    |   movel(p[0.416217, -0.000852, -0.000100, 0.000000, -3.141593, 0.000000],accel_mss,speed_ms,0,blend_radius_m)
    |   movel(p[0.416898, -0.000524, -0.000100, 0.000000, -3.141593, 0.000000],accel_mss,speed_ms,0,blend_radius_m)
    |   movel(p[0.417586, -0.000221, -0.000100, 0.000000, 3.141593, 0.000000],accel_mss,speed_ms,0,blend_radius_m)
    |   movel(p[0.417752, -0.000150, -0.000100, 0.000000, -3.141593, 0.000000],accel_mss,speed_ms,0,0.000)
    |   movel(p[0.418040, -0.000026, -0.000100, 0.000000, -3.141593, 0.000000],accel_mss,speed_ms,0,0.000)
    |   movel(p[0.418373, 0.000118, -0.000100, 0.000000, -3.141593, 0.000000],accel_mss,speed_ms,0,0.000)
    |   movel(p[0.418711, 0.000265, -0.000100, 0.000000, -3.141593, 0.000000],accel_mss,speed_ms,0,0.000)
    |   movel(p[0.419555, 0.000597, -0.000100, 0.000000, -3.141593, 0.000000],accel_mss,speed_ms,0,blend_radius_m)
    |   movel(p[0.420567, 0.000924, -0.000100, 0.000000, 3.141593, 0.000000],accel_mss,speed_ms,0,blend_radius_m)
    |   movel(p[0.421755, 0.001251, -0.000100, 0.000000, -3.141593, 0.000000],accel_mss,speed_ms,0,blend_radius_m)
    |   movel(p[0.423136, 0.001581, -0.000100, 0.000000, -3.141593, 0.000000],accel_mss,speed_ms,0,blend_radius_m)
    |   movel(p[0.424710, 0.001831, -0.000100, 0.000000, 3.141593, 0.000000],accel_mss,speed_ms,0,blend_radius_m)
    |   movel(p[0.426559, 0.001928, -0.000100, 0.000000, 3.141593, 0.000000],accel_mss,speed_ms,0,blend_radius_m)
    |   movel(p[0.428336, 0.001876, -0.000100, 0.000000, -3.141593, 0.000000],accel_mss,speed_ms,0,blend_radius_m)
    |   movel(p[0.429661, 0.001658, -0.000100, 0.000000, -3.141593, 0.000000],accel_mss,speed_ms,0,blend_radius_m)
    |   movel(p[0.430073, 0.001550, -0.000100, 0.000000, -3.141593, 0.000000],accel_mss,speed_ms,0,0.000)
    |   movel(p[0.430504, 0.001438, -0.000100, 0.000000, 3.141593, 0.000000],accel_mss,speed_ms,0,0.000)
    |   movel(p[0.430895, 0.001337, -0.000100, 0.000000, -3.141593, 0.000000],accel_mss,speed_ms,0,0.000)
    |   movel(p[0.431163, 0.001269, -0.000100, 0.000000, -3.141593, 0.000000],accel_mss,speed_ms,0,0.000)
    |   movel(p[0.432181, 0.000939, -0.000100, 0.000000, -3.141593, 0.000000],accel_mss,speed_ms,0,blend_radius_m)
    |   movel(p[0.433399, 0.000403, -0.000100, 0.000000, -3.141593, 0.000000],accel_mss,speed_ms,0,blend_radius_m)
    |   movel(p[0.434515, -0.000180, -0.000100, 0.000000, 3.141593, 0.000000],accel_mss,speed_ms,0,blend_radius_m)
    |   movel(p[0.435077, -0.000621, -0.000100, 0.000000, 3.141593, 0.000000],accel_mss,speed_ms,0,blend_radius_m)
    |   movel(p[0.435218, -0.000758, -0.000100, 0.000000, -3.141593, 0.000000],accel_mss,speed_ms,0,0.000)
    |   movel(p[0.435364, -0.000873, -0.000100, 0.000000, -3.141593, 0.000000],accel_mss,speed_ms,0,0.000)
    |   movel(p[0.435496, -0.000956, -0.000100, 0.000000, 3.141593, 0.000000],accel_mss,speed_ms,0,0.000)
    |   movel(p[0.435800, -0.001069, -0.000100, 0.000000, -3.141593, 0.000000],accel_mss,speed_ms,0,0.000)
    |   movel(p[0.437336, -0.002626, -0.000100, 0.000000, -3.141593, 0.000000],accel_mss,speed_ms,0,blend_radius_m)
    |   movel(p[0.438726, -0.004069, -0.000100, 0.000000, -3.141593, 0.000000],accel_mss,speed_ms,0,blend_radius_m)
    |   movel(p[0.439357, -0.004825, -0.000100, 0.000000, -3.141593, 0.000000],accel_mss,speed_ms,0,blend_radius_m)
    |   movel(p[0.439502, -0.005031, -0.000100, 0.000000, 3.141593, 0.000000],accel_mss,speed_ms,0,0.000)
    |   movel(p[0.439674, -0.005293, -0.000100, 0.000000, -3.141593, 0.000000],accel_mss,speed_ms,0,0.000)
    |   movel(p[0.439844, -0.005566, -0.000100, 0.000000, 3.141593, 0.000000],accel_mss,speed_ms,0,0.000)
    |   movel(p[0.439984, -0.005806, -0.000100, 0.000000, -3.141593, 0.000000],accel_mss,speed_ms,0,0.000)
    |   movel(p[0.440137, -0.006078, -0.000100, 0.000000, -3.141593, 0.000000],accel_mss,speed_ms,0,0.000)
    |   movel(p[0.440290, -0.006350, -0.000100, 0.000000, 3.141593, 0.000000],accel_mss,speed_ms,0,0.000)
    |   movel(p[0.439826, -0.006519, -0.000100, 0.000000, -3.141593, 0.000000],accel_mss,speed_ms,0,0.000)
    |   movel(p[0.439363, -0.006689, -0.000100, 0.000000, -3.141593, 0.000000],accel_mss,speed_ms,0,0.000)
    |   movel(p[0.437743, -0.007355, -0.000100, 0.000000, 3.141593, 0.000000],accel_mss,speed_ms,0,blend_radius_m)
    |   movel(p[0.436100, -0.008178, -0.000100, 0.000000, -3.141593, 0.000000],accel_mss,speed_ms,0,blend_radius_m)
    |   movel(p[0.434697, -0.009002, -0.000100, 0.000000, -3.141593, 0.000000],accel_mss,speed_ms,0,blend_radius_m)
    |   movel(p[0.434010, -0.009605, -0.000100, 0.000000, -3.141593, 0.000000],accel_mss,speed_ms,0,blend_radius_m)
    |   movel(p[0.433927, -0.009690, -0.000100, 0.000000, -3.141593, 0.000000],accel_mss,speed_ms,0,0.000)
    |   movel(p[0.433830, -0.009763, -0.000100, 0.000000, -3.141593, 0.000000],accel_mss,speed_ms,0,0.000)
    |   movel(p[0.433736, -0.009813, -0.000100, 0.000000, -3.141593, 0.000000],accel_mss,speed_ms,0,0.000)
    |   movel(p[0.433418, -0.009924, -0.000100, 0.000000, -3.141593, 0.000000],accel_mss,speed_ms,0,0.000)
    |   movel(p[0.432629, -0.010689, -0.000100, 0.000000, 3.141593, 0.000000],accel_mss,speed_ms,0,blend_radius_m)
    |   movel(p[0.431857, -0.011472, -0.000100, 0.000000, -3.141593, 0.000000],accel_mss,speed_ms,0,blend_radius_m)
    |   movel(p[0.431761, -0.011710, -0.000100, 0.000000, -3.141593, 0.000000],accel_mss,speed_ms,0,0.000)
    |   movel(p[0.431651, -0.011931, -0.000100, 0.000000, -3.141593, 0.000000],accel_mss,speed_ms,0,0.000)
    |   movel(p[0.431530, -0.012081, -0.000100, 0.000000, -3.141593, 0.000000],accel_mss,speed_ms,0,0.000)
    |   movel(p[0.431386, -0.012228, -0.000100, 0.000000, -3.141593, 0.000000],accel_mss,speed_ms,0,0.000)
    |   movel(p[0.431242, -0.012373, -0.000100, 0.000000, -3.141593, 0.000000],accel_mss,speed_ms,0,0.000)
    |   movel(p[0.431121, -0.012518, -0.000100, 0.000000, -3.141593, 0.000000],accel_mss,speed_ms,0,0.000)
    |   movel(p[0.431032, -0.012645, -0.000100, 0.000000, -3.141593, 0.000000],accel_mss,speed_ms,0,0.000)
    |   movel(p[0.430995, -0.012795, -0.000100, 0.000000, -3.141593, 0.000000],accel_mss,speed_ms,0,0.000)
    |   movel(p[0.430928, -0.012933, -0.000100, 0.000000, 3.141593, 0.000000],accel_mss,speed_ms,0,0.000)
    |   movel(p[0.430837, -0.013093, -0.000100, 0.000000, -3.141593, 0.000000],accel_mss,speed_ms,0,0.000)
    |   movel(p[0.430728, -0.013255, -0.000100, 0.000000, -3.141593, 0.000000],accel_mss,speed_ms,0,0.000)
    |   movel(p[0.430595, -0.013484, -0.000100, 0.000000, -3.141593, 0.000000],accel_mss,speed_ms,0,0.000)
    |   movel(p[0.430417, -0.013889, -0.000100, 0.000000, -3.141593, 0.000000],accel_mss,speed_ms,0,0.000)
    |   movel(p[0.430232, -0.014365, -0.000100, 0.000000, -3.141593, 0.000000],accel_mss,speed_ms,0,blend_radius_m)
    |   movel(p[0.430065, -0.014853, -0.000100, 0.000000, -3.141593, 0.000000],accel_mss,speed_ms,0,blend_radius_m)
    |   movel(p[0.429860, -0.015581, -0.000100, 0.000000, 3.141593, 0.000000],accel_mss,speed_ms,0,blend_radius_m)
    |   movel(p[0.429754, -0.016174, -0.000100, 0.000000, 3.141593, 0.000000],accel_mss,speed_ms,0,blend_radius_m)
    |   movel(p[0.429710, -0.016862, -0.000100, 0.000000, 3.141593, 0.000000],accel_mss,speed_ms,0,blend_radius_m)
    |   movel(p[0.429711, -0.017960, -0.000100, 0.000000, -3.141593, 0.000000],accel_mss,speed_ms,0,blend_radius_m)
    |   movel(p[0.429734, -0.018811, -0.000100, 0.000000, 3.141593, 0.000000],accel_mss,speed_ms,0,blend_radius_m)
    |   movel(p[0.429778, -0.019434, -0.000100, 0.000000, -3.141593, 0.000000],accel_mss,speed_ms,0,blend_radius_m)
    |   movel(p[0.429837, -0.019884, -0.000100, 0.000000, -3.141593, 0.000000],accel_mss,speed_ms,0,0.000)
    |   movel(p[0.429922, -0.020049, -0.000100, 0.000000, 3.141593, 0.000000],accel_mss,speed_ms,0,0.000)
    |   movel(p[0.430062, -0.020114, -0.000100, 0.000000, -3.141593, 0.000000],accel_mss,speed_ms,0,0.000)
    |   movel(p[0.430262, -0.020097, -0.000100, 0.000000, 3.141593, 0.000000],accel_mss,speed_ms,0,0.000)
    |   movel(p[0.430563, -0.019991, -0.000100, 0.000000, -3.141593, 0.000000],accel_mss,speed_ms,0,0.000)
    |   movel(p[0.431055, -0.019755, -0.000100, 0.000000, -3.141593, 0.000000],accel_mss,speed_ms,0,blend_radius_m)
    |   movel(p[0.431427, -0.019573, -0.000100, 0.000000, -3.141593, 0.000000],accel_mss,speed_ms,0,0.000)
    |   movel(p[0.431760, -0.019418, -0.000100, 0.000000, -3.141593, 0.000000],accel_mss,speed_ms,0,0.000)
    |   movel(p[0.432042, -0.019295, -0.000100, 0.000000, -3.141593, 0.000000],accel_mss,speed_ms,0,0.000)
    |   movel(p[0.432189, -0.019263, -0.000100, 0.000000, -3.141593, 0.000000],accel_mss,speed_ms,0,0.000)
    |   movel(p[0.432322, -0.019196, -0.000100, 0.000000, 3.141593, 0.000000],accel_mss,speed_ms,0,0.000)
    |   movel(p[0.432477, -0.019106, -0.000100, 0.000000, 3.141593, 0.000000],accel_mss,speed_ms,0,0.000)
    |   movel(p[0.432638, -0.018999, -0.000100, 0.000000, -3.141593, 0.000000],accel_mss,speed_ms,0,0.000)
    |   movel(p[0.432833, -0.018877, -0.000100, 0.000000, 3.141593, 0.000000],accel_mss,speed_ms,0,0.000)
    |   movel(p[0.433095, -0.018742, -0.000100, 0.000000, -3.141593, 0.000000],accel_mss,speed_ms,0,0.000)
    |   movel(p[0.433377, -0.018615, -0.000100, 0.000000, 3.141593, 0.000000],accel_mss,speed_ms,0,0.000)
    |   movel(p[0.433636, -0.018517, -0.000100, 0.000000, 3.141593, 0.000000],accel_mss,speed_ms,0,0.000)
    |   movel(p[0.433877, -0.018432, -0.000100, 0.000000, -3.141593, 0.000000],accel_mss,speed_ms,0,0.000)
    |   movel(p[0.434105, -0.018343, -0.000100, 0.000000, 3.141593, 0.000000],accel_mss,speed_ms,0,0.000)
    |   movel(p[0.434295, -0.018261, -0.000100, 0.000000, -3.141593, 0.000000],accel_mss,speed_ms,0,0.000)
    |   movel(p[0.434389, -0.018208, -0.000100, 0.000000, -3.141593, 0.000000],accel_mss,speed_ms,0,0.000)
    |   movel(p[0.434943, -0.017924, -0.000100, 0.000000, -3.141593, 0.000000],accel_mss,speed_ms,0,blend_radius_m)
    |   movel(p[0.436858, -0.017281, -0.000100, 0.000000, -3.141593, 0.000000],accel_mss,speed_ms,0,blend_radius_m)
    |   movel(p[0.438844, -0.016659, -0.000100, 0.000000, 3.141593, 0.000000],accel_mss,speed_ms,0,blend_radius_m)
    |   movel(p[0.440461, -0.016220, -0.000100, 0.000000, -3.141593, 0.000000],accel_mss,speed_ms,0,blend_radius_m)
    |   movel(p[0.443462, -0.015545, -0.000100, 0.000000, -3.141593, 0.000000],accel_mss,speed_ms,0,blend_radius_m)
    |   movel(p[0.445689, -0.015200, -0.000100, 0.000000, -3.141593, 0.000000],accel_mss,speed_ms,0,blend_radius_m)
    |   movel(p[0.448089, -0.015048, -0.000100, 0.000000, 3.141593, 0.000000],accel_mss,speed_ms,0,blend_radius_m)
    |   movel(p[0.451786, -0.015019, -0.000100, 0.000000, -3.141593, 0.000000],accel_mss,speed_ms,0,blend_radius_m)
    |   movel(p[0.454871, -0.015067, -0.000100, 0.000000, -3.141593, 0.000000],accel_mss,speed_ms,0,blend_radius_m)
    |   movel(p[0.456835, -0.015196, -0.000100, 0.000000, 3.141593, 0.000000],accel_mss,speed_ms,0,blend_radius_m)
    |   movel(p[0.458642, -0.015468, -0.000100, 0.000000, -3.141593, 0.000000],accel_mss,speed_ms,0,blend_radius_m)
    |   movel(p[0.461086, -0.015994, -0.000100, 0.000000, -3.141593, 0.000000],accel_mss,speed_ms,0,blend_radius_m)
    |   movel(p[0.462544, -0.016380, -0.000100, 0.000000, -3.141593, 0.000000],accel_mss,speed_ms,0,blend_radius_m)
    |   movel(p[0.464600, -0.017008, -0.000100, 0.000000, -3.141593, 0.000000],accel_mss,speed_ms,0,blend_radius_m)
    |   movel(p[0.466617, -0.017663, -0.000100, 0.000000, -3.141593, 0.000000],accel_mss,speed_ms,0,blend_radius_m)
    |   movel(p[0.467386, -0.017990, -0.000100, 0.000000, 3.141593, 0.000000],accel_mss,speed_ms,0,blend_radius_m)
    |   movel(p[0.467568, -0.018081, -0.000100, 0.000000, -3.141593, 0.000000],accel_mss,speed_ms,0,0.000)
    |   movel(p[0.467741, -0.018157, -0.000100, 0.000000, -3.141593, 0.000000],accel_mss,speed_ms,0,0.000)
    |   movel(p[0.467889, -0.018214, -0.000100, 0.000000, 3.141593, 0.000000],accel_mss,speed_ms,0,0.000)
    |   movel(p[0.468168, -0.018270, -0.000100, 0.000000, -3.141593, 0.000000],accel_mss,speed_ms,0,0.000)
    |   movel(p[0.468732, -0.018516, -0.000100, 0.000000, -3.141593, 0.000000],accel_mss,speed_ms,0,blend_radius_m)
    |   movel(p[0.469521, -0.018887, -0.000100, 0.000000, -3.141593, 0.000000],accel_mss,speed_ms,0,blend_radius_m)
    |   movel(p[0.470686, -0.019461, -0.000100, 0.000000, -3.141593, 0.000000],accel_mss,speed_ms,0,blend_radius_m)
    |   movel(p[0.472327, -0.020285, -0.000100, 0.000000, -3.141593, 0.000000],accel_mss,speed_ms,0,blend_radius_m)
    |   movel(p[0.473356, -0.020827, -0.000100, 0.000000, -3.141593, 0.000000],accel_mss,speed_ms,0,blend_radius_m)
    |   movel(p[0.474059, -0.021232, -0.000100, 0.000000, -3.141593, 0.000000],accel_mss,speed_ms,0,blend_radius_m)
    |   movel(p[0.474563, -0.021575, -0.000100, 0.000000, 3.141593, 0.000000],accel_mss,speed_ms,0,blend_radius_m)
    |   movel(p[0.474775, -0.021730, -0.000100, 0.000000, -3.141593, 0.000000],accel_mss,speed_ms,0,0.000)
    |   movel(p[0.474976, -0.021860, -0.000100, 0.000000, 3.141593, 0.000000],accel_mss,speed_ms,0,0.000)
    |   movel(p[0.475148, -0.021958, -0.000100, 0.000000, -3.141593, 0.000000],accel_mss,speed_ms,0,0.000)
    |   movel(p[0.475298, -0.021997, -0.000100, 0.000000, -3.141593, 0.000000],accel_mss,speed_ms,0,0.000)
    |   movel(p[0.475404, -0.022066, -0.000100, 0.000000, -3.141593, 0.000000],accel_mss,speed_ms,0,0.000)
    |   movel(p[0.475522, -0.022164, -0.000100, 0.000000, -3.141593, 0.000000],accel_mss,speed_ms,0,0.000)
    |   movel(p[0.475636, -0.022278, -0.000100, 0.000000, -3.141593, 0.000000],accel_mss,speed_ms,0,0.000)
    |   movel(p[0.475753, -0.022393, -0.000100, 0.000000, 3.141593, 0.000000],accel_mss,speed_ms,0,0.000)
    |   movel(p[0.475880, -0.022490, -0.000100, 0.000000, -3.141593, 0.000000],accel_mss,speed_ms,0,0.000)
    |   movel(p[0.475999, -0.022558, -0.000100, 0.000000, -3.141593, 0.000000],accel_mss,speed_ms,0,0.000)
    |   movel(p[0.476173, -0.022598, -0.000100, 0.000000, -3.141593, 0.000000],accel_mss,speed_ms,0,0.000)
    |   movel(p[0.476292, -0.022666, -0.000100, 0.000000, -3.141593, 0.000000],accel_mss,speed_ms,0,0.000)
    |   movel(p[0.476419, -0.022764, -0.000100, 0.000000, 3.141593, 0.000000],accel_mss,speed_ms,0,0.000)
    |   movel(p[0.476536, -0.022878, -0.000100, 0.000000, 3.141593, 0.000000],accel_mss,speed_ms,0,0.000)
    |   movel(p[0.476651, -0.022993, -0.000100, 0.000000, -3.141593, 0.000000],accel_mss,speed_ms,0,0.000)
    |   movel(p[0.476771, -0.023090, -0.000100, 0.000000, 3.141593, 0.000000],accel_mss,speed_ms,0,0.000)
    |   movel(p[0.476880, -0.023159, -0.000100, 0.000000, -3.141593, 0.000000],accel_mss,speed_ms,0,0.000)
    |   movel(p[0.477050, -0.023211, -0.000100, 0.000000, -3.141593, 0.000000],accel_mss,speed_ms,0,0.000)
    |   movel(p[0.477427, -0.023513, -0.000100, 0.000000, -3.141593, 0.000000],accel_mss,speed_ms,0,0.000)
    |   movel(p[0.477865, -0.023881, -0.000100, 0.000000, -3.141593, 0.000000],accel_mss,speed_ms,0,blend_radius_m)
    |   movel(p[0.478356, -0.024317, -0.000100, 0.000000, -3.141593, 0.000000],accel_mss,speed_ms,0,blend_radius_m)
    |   movel(p[0.478838, -0.024746, -0.000100, 0.000000, -3.141593, 0.000000],accel_mss,speed_ms,0,blend_radius_m)
    |   movel(p[0.479242, -0.025085, -0.000100, 0.000000, 3.141593, 0.000000],accel_mss,speed_ms,0,blend_radius_m)
    |   movel(p[0.479575, -0.025349, -0.000100, 0.000000, 3.141593, 0.000000],accel_mss,speed_ms,0,0.000)
    |   movel(p[0.480294, -0.025926, -0.000100, 0.000000, -3.141593, 0.000000],accel_mss,speed_ms,0,blend_radius_m)
    |   movel(p[0.481044, -0.026647, -0.000100, 0.000000, -3.141593, 0.000000],accel_mss,speed_ms,0,blend_radius_m)
    |   movel(p[0.481936, -0.027528, -0.000100, 0.000000, -3.141593, 0.000000],accel_mss,speed_ms,0,blend_radius_m)
    |   movel(p[0.482827, -0.028427, -0.000100, 0.000000, -3.141593, 0.000000],accel_mss,speed_ms,0,blend_radius_m)
    |   movel(p[0.483578, -0.029205, -0.000100, 0.000000, -3.141593, 0.000000],accel_mss,speed_ms,0,blend_radius_m)
    |   movel(p[0.484227, -0.029891, -0.000100, 0.000000, 3.141593, 0.000000],accel_mss,speed_ms,0,blend_radius_m)
    |   movel(p[0.484290, -0.030061, -0.000100, 0.000000, -3.141593, 0.000000],accel_mss,speed_ms,0,0.000)
    |   movel(p[0.484569, -0.030409, -0.000100, 0.000000, 3.141593, 0.000000],accel_mss,speed_ms,0,0.000)
    |   movel(p[0.484909, -0.030813, -0.000100, 0.000000, -3.141593, 0.000000],accel_mss,speed_ms,0,blend_radius_m)
    |   movel(p[0.485311, -0.031268, -0.000100, 0.000000, -3.141593, 0.000000],accel_mss,speed_ms,0,blend_radius_m)
    |   movel(p[0.485713, -0.031725, -0.000100, 0.000000, -3.141593, 0.000000],accel_mss,speed_ms,0,blend_radius_m)
    |   movel(p[0.486053, -0.032134, -0.000100, 0.000000, -3.141593, 0.000000],accel_mss,speed_ms,0,blend_radius_m)
    |   movel(p[0.486328, -0.032485, -0.000100, 0.000000, -3.141593, 0.000000],accel_mss,speed_ms,0,0.000)
    |   movel(p[0.486361, -0.032581, -0.000100, 0.000000, 3.141593, 0.000000],accel_mss,speed_ms,0,0.000)
    |   movel(p[0.486449, -0.032767, -0.000100, 0.000000, -3.141593, 0.000000],accel_mss,speed_ms,0,0.000)
    |   movel(p[0.486546, -0.032888, -0.000100, 0.000000, -3.141593, 0.000000],accel_mss,speed_ms,0,0.000)
    |   movel(p[0.486661, -0.033003, -0.000100, 0.000000, -3.141593, 0.000000],accel_mss,speed_ms,0,0.000)
    |   movel(p[0.486776, -0.033120, -0.000100, 0.000000, 3.141593, 0.000000],accel_mss,speed_ms,0,0.000)
    |   movel(p[0.486873, -0.033248, -0.000100, 0.000000, -3.141593, 0.000000],accel_mss,speed_ms,0,0.000)
    |   movel(p[0.486941, -0.033366, -0.000100, 0.000000, -3.141593, 0.000000],accel_mss,speed_ms,0,0.000)
    |   movel(p[0.486981, -0.033540, -0.000100, 0.000000, -3.141593, 0.000000],accel_mss,speed_ms,0,0.000)
    |   movel(p[0.487049, -0.033659, -0.000100, 0.000000, -3.141593, 0.000000],accel_mss,speed_ms,0,0.000)
    |   movel(p[0.487146, -0.033786, -0.000100, 0.000000, -3.141593, 0.000000],accel_mss,speed_ms,0,0.000)
    |   movel(p[0.487261, -0.033903, -0.000100, 0.000000, -3.141593, 0.000000],accel_mss,speed_ms,0,0.000)
    |   movel(p[0.487376, -0.034018, -0.000100, 0.000000, -3.141593, 0.000000],accel_mss,speed_ms,0,0.000)
    |   movel(p[0.487473, -0.034137, -0.000100, 0.000000, -3.141593, 0.000000],accel_mss,speed_ms,0,0.000)
    |   movel(p[0.487542, -0.034245, -0.000100, 0.000000, -3.141593, 0.000000],accel_mss,speed_ms,0,0.000)
    |   movel(p[0.487582, -0.034401, -0.000100, 0.000000, -3.141593, 0.000000],accel_mss,speed_ms,0,0.000)
    |   movel(p[0.487682, -0.034579, -0.000100, 0.000000, -3.141593, 0.000000],accel_mss,speed_ms,0,0.000)
    |   movel(p[0.487815, -0.034787, -0.000100, 0.000000, -3.141593, 0.000000],accel_mss,speed_ms,0,0.000)
    |   movel(p[0.487973, -0.035007, -0.000100, 0.000000, -3.141593, 0.000000],accel_mss,speed_ms,0,0.000)
    |   movel(p[0.488406, -0.035609, -0.000100, 0.000000, -3.141593, 0.000000],accel_mss,speed_ms,0,blend_radius_m)
    |   movel(p[0.488726, -0.036121, -0.000100, 0.000000, -3.141593, 0.000000],accel_mss,speed_ms,0,blend_radius_m)
    |   movel(p[0.488944, -0.036553, -0.000100, 0.000000, -3.141593, 0.000000],accel_mss,speed_ms,0,0.000)
    |   movel(p[0.489054, -0.036903, -0.000100, 0.000000, -3.141593, 0.000000],accel_mss,speed_ms,0,0.000)
    |   movel(p[0.489130, -0.037075, -0.000100, 0.000000, -3.141593, 0.000000],accel_mss,speed_ms,0,0.000)
    |   movel(p[0.489199, -0.037181, -0.000100, 0.000000, -3.141593, 0.000000],accel_mss,speed_ms,0,0.000)
    |   movel(p[0.489274, -0.037278, -0.000100, 0.000000, -3.141593, 0.000000],accel_mss,speed_ms,0,0.000)
    |   movel(p[0.489617, -0.037792, -0.000100, 0.000000, -3.141593, 0.000000],accel_mss,speed_ms,0,blend_radius_m)
    |   movel(p[0.490361, -0.039291, -0.000100, 0.000000, -3.141593, 0.000000],accel_mss,speed_ms,0,blend_radius_m)
    |   movel(p[0.491079, -0.040819, -0.000100, 0.000000, -3.141593, 0.000000],accel_mss,speed_ms,0,blend_radius_m)
    |   movel(p[0.491523, -0.041907, -0.000100, 0.000000, -3.141593, 0.000000],accel_mss,speed_ms,0,blend_radius_m)
    |   movel(p[0.492063, -0.043418, -0.000100, 0.000000, -3.141593, 0.000000],accel_mss,speed_ms,0,blend_radius_m)
    |   movel(p[0.492524, -0.044767, -0.000100, 0.000000, -3.141593, 0.000000],accel_mss,speed_ms,0,blend_radius_m)
    |   movel(p[0.492955, -0.046099, -0.000100, 0.000000, -3.141593, 0.000000],accel_mss,speed_ms,0,blend_radius_m)
    |   movel(p[0.493401, -0.047553, -0.000100, 0.000000, -3.141593, 0.000000],accel_mss,speed_ms,0,blend_radius_m)
    |   movel(p[0.493523, -0.048000, -0.000100, 0.000000, -3.141593, 0.000000],accel_mss,speed_ms,0,0.000)
    |   movel(p[0.493636, -0.048500, -0.000100, 0.000000, -3.141593, 0.000000],accel_mss,speed_ms,0,blend_radius_m)
    |   movel(p[0.493728, -0.048991, -0.000100, 0.000000, -3.141593, 0.000000],accel_mss,speed_ms,0,0.000)
    |   movel(p[0.493784, -0.049411, -0.000100, 0.000000, -3.141593, 0.000000],accel_mss,speed_ms,0,0.000)
    |   movel(p[0.493817, -0.049655, -0.000100, 0.000000, -3.141593, 0.000000],accel_mss,speed_ms,0,0.000)
    |   movel(p[0.493908, -0.050217, -0.000100, 0.000000, 3.141593, 0.000000],accel_mss,speed_ms,0,blend_radius_m)
    |   movel(p[0.494021, -0.050885, -0.000100, 0.000000, -3.141593, 0.000000],accel_mss,speed_ms,0,blend_radius_m)
    |   movel(p[0.494147, -0.051603, -0.000100, 0.000000, -3.141593, 0.000000],accel_mss,speed_ms,0,blend_radius_m)
    |   movel(p[0.494558, -0.054697, -0.000100, 0.000000, 3.141593, 0.000000],accel_mss,speed_ms,0,blend_radius_m)
    |   movel(p[0.494697, -0.057850, -0.000100, 0.000000, 3.141593, 0.000000],accel_mss,speed_ms,0,blend_radius_m)
    |   movel(p[0.494562, -0.061080, -0.000100, 0.000000, -3.141593, 0.000000],accel_mss,speed_ms,0,blend_radius_m)
    |   movel(p[0.494155, -0.064404, -0.000100, 0.000000, -3.141593, 0.000000],accel_mss,speed_ms,0,blend_radius_m)
    |   movel(p[0.494041, -0.065118, -0.000100, 0.000000, -3.141593, 0.000000],accel_mss,speed_ms,0,blend_radius_m)
    |   movel(p[0.493930, -0.065816, -0.000100, 0.000000, -3.141593, 0.000000],accel_mss,speed_ms,0,blend_radius_m)
    |   movel(p[0.493836, -0.066416, -0.000100, 0.000000, -3.141593, 0.000000],accel_mss,speed_ms,0,blend_radius_m)
    |   movel(p[0.493784, -0.066753, -0.000100, 0.000000, -3.141593, 0.000000],accel_mss,speed_ms,0,0.000)
    |   movel(p[0.493465, -0.068250, -0.000100, 0.000000, -3.141593, 0.000000],accel_mss,speed_ms,0,blend_radius_m)
    |   movel(p[0.492719, -0.070782, -0.000100, 0.000000, -3.141593, 0.000000],accel_mss,speed_ms,0,blend_radius_m)
    |   movel(p[0.491886, -0.073338, -0.000100, 0.000000, -3.141593, 0.000000],accel_mss,speed_ms,0,blend_radius_m)
    |   movel(p[0.491207, -0.075078, -0.000100, 0.000000, -3.141593, 0.000000],accel_mss,speed_ms,0,blend_radius_m)
    |   movel(p[0.491058, -0.075416, -0.000100, 0.000000, -3.141593, 0.000000],accel_mss,speed_ms,0,0.000)
    |   movel(p[0.490913, -0.075749, -0.000100, 0.000000, -3.141593, 0.000000],accel_mss,speed_ms,0,0.000)
    |   movel(p[0.490787, -0.076037, -0.000100, 0.000000, -3.141593, 0.000000],accel_mss,speed_ms,0,0.000)
    |   movel(p[0.490715, -0.076203, -0.000100, 0.000000, -3.141593, 0.000000],accel_mss,speed_ms,0,0.000)
    |   movel(p[0.490443, -0.076801, -0.000100, 0.000000, -3.141593, 0.000000],accel_mss,speed_ms,0,blend_radius_m)
    |   movel(p[0.490066, -0.077573, -0.000100, 0.000000, -3.141593, 0.000000],accel_mss,speed_ms,0,blend_radius_m)
    |   movel(p[0.489660, -0.078369, -0.000100, 0.000000, -3.141593, 0.000000],accel_mss,speed_ms,0,blend_radius_m)
    |   movel(p[0.489292, -0.079053, -0.000100, 0.000000, 3.141593, 0.000000],accel_mss,speed_ms,0,blend_radius_m)
    |   movel(p[0.489070, -0.079458, -0.000100, 0.000000, -3.141593, 0.000000],accel_mss,speed_ms,0,0.000)
    |   movel(p[0.488816, -0.079931, -0.000100, 0.000000, -3.141593, 0.000000],accel_mss,speed_ms,0,blend_radius_m)
    |   movel(p[0.488569, -0.080398, -0.000100, 0.000000, -3.141593, 0.000000],accel_mss,speed_ms,0,blend_radius_m)
    |   movel(p[0.488372, -0.080778, -0.000100, 0.000000, -3.141593, 0.000000],accel_mss,speed_ms,0,0.000)
    |   movel(p[0.488175, -0.081139, -0.000100, 0.000000, -3.141593, 0.000000],accel_mss,speed_ms,0,0.000)
    |   movel(p[0.487930, -0.081542, -0.000100, 0.000000, -3.141593, 0.000000],accel_mss,speed_ms,0,0.000)
    |   movel(p[0.487677, -0.081924, -0.000100, 0.000000, -3.141593, 0.000000],accel_mss,speed_ms,0,0.000)
    |   movel(p[0.487457, -0.082219, -0.000100, 0.000000, -3.141593, 0.000000],accel_mss,speed_ms,0,0.000)
    |   movel(p[0.487267, -0.082465, -0.000100, 0.000000, -3.141593, 0.000000],accel_mss,speed_ms,0,0.000)
    |   movel(p[0.487107, -0.082696, -0.000100, 0.000000, -3.141593, 0.000000],accel_mss,speed_ms,0,0.000)
    |   movel(p[0.486985, -0.082893, -0.000100, 0.000000, -3.141593, 0.000000],accel_mss,speed_ms,0,0.000)
    |   movel(p[0.486939, -0.083057, -0.000100, 0.000000, -3.141593, 0.000000],accel_mss,speed_ms,0,0.000)
    |   movel(p[0.486851, -0.083187, -0.000100, 0.000000, -3.141593, 0.000000],accel_mss,speed_ms,0,0.000)
    |   movel(p[0.486730, -0.083333, -0.000100, 0.000000, -3.141593, 0.000000],accel_mss,speed_ms,0,0.000)
    |   movel(p[0.486586, -0.083478, -0.000100, 0.000000, -3.141593, 0.000000],accel_mss,speed_ms,0,0.000)
    |   movel(p[0.486442, -0.083626, -0.000100, 0.000000, -3.141593, 0.000000],accel_mss,speed_ms,0,0.000)
    |   movel(p[0.486321, -0.083779, -0.000100, 0.000000, -3.141593, 0.000000],accel_mss,speed_ms,0,0.000)
    |   movel(p[0.486234, -0.083916, -0.000100, 0.000000, -3.141593, 0.000000],accel_mss,speed_ms,0,0.000)
    |   movel(p[0.486191, -0.084092, -0.000100, 0.000000, -3.141593, 0.000000],accel_mss,speed_ms,0,0.000)
    |   movel(p[0.486123, -0.084210, -0.000100, 0.000000, -3.141593, 0.000000],accel_mss,speed_ms,0,0.000)
    |   movel(p[0.486026, -0.084337, -0.000100, 0.000000, -3.141593, 0.000000],accel_mss,speed_ms,0,0.000)
    |   movel(p[0.485911, -0.084453, -0.000100, 0.000000, -3.141593, 0.000000],accel_mss,speed_ms,0,0.000)
    |   movel(p[0.485796, -0.084568, -0.000100, 0.000000, -3.141593, 0.000000],accel_mss,speed_ms,0,0.000)
    |   movel(p[0.485699, -0.084689, -0.000100, 0.000000, -3.141593, 0.000000],accel_mss,speed_ms,0,0.000)
    |   movel(p[0.485630, -0.084799, -0.000100, 0.000000, -3.141593, 0.000000],accel_mss,speed_ms,0,0.000)
    |   movel(p[0.485577, -0.084972, -0.000100, 0.000000, -3.141593, 0.000000],accel_mss,speed_ms,0,0.000)
    |   movel(p[0.485258, -0.085366, -0.000100, 0.000000, -3.141593, 0.000000],accel_mss,speed_ms,0,blend_radius_m)
    |   movel(p[0.484871, -0.085823, -0.000100, 0.000000, -3.141593, 0.000000],accel_mss,speed_ms,0,blend_radius_m)
    |   movel(p[0.484411, -0.086337, -0.000100, 0.000000, -3.141593, 0.000000],accel_mss,speed_ms,0,blend_radius_m)
    |   movel(p[0.483951, -0.086850, -0.000100, 0.000000, -3.141593, 0.000000],accel_mss,speed_ms,0,blend_radius_m)
    |   movel(p[0.483563, -0.087301, -0.000100, 0.000000, -3.141593, 0.000000],accel_mss,speed_ms,0,blend_radius_m)
    |   movel(p[0.483240, -0.087692, -0.000100, 0.000000, -3.141593, 0.000000],accel_mss,speed_ms,0,blend_radius_m)
    |   movel(p[0.483129, -0.087975, -0.000100, 0.000000, -3.141593, 0.000000],accel_mss,speed_ms,0,0.000)
    |   movel(p[0.481598, -0.089513, -0.000100, 0.000000, -3.141593, 0.000000],accel_mss,speed_ms,0,blend_radius_m)
    |   movel(p[0.480062, -0.091046, -0.000100, 0.000000, -3.141593, 0.000000],accel_mss,speed_ms,0,blend_radius_m)
    |   movel(p[0.479862, -0.091128, -0.000100, 0.000000, -3.141593, 0.000000],accel_mss,speed_ms,0,0.000)
    |   movel(p[0.479385, -0.091481, -0.000100, 0.000000, -3.141593, 0.000000],accel_mss,speed_ms,0,blend_radius_m)
    |   movel(p[0.478932, -0.091868, -0.000100, 0.000000, -3.141593, 0.000000],accel_mss,speed_ms,0,blend_radius_m)
    |   movel(p[0.478420, -0.092328, -0.000100, 0.000000, -3.141593, 0.000000],accel_mss,speed_ms,0,blend_radius_m)
    |   movel(p[0.477906, -0.092788, -0.000100, 0.000000, -3.141593, 0.000000],accel_mss,speed_ms,0,blend_radius_m)
    |   movel(p[0.477449, -0.093176, -0.000100, 0.000000, -3.141593, 0.000000],accel_mss,speed_ms,0,blend_radius_m)
    |   movel(p[0.477054, -0.093494, -0.000100, 0.000000, -3.141593, 0.000000],accel_mss,speed_ms,0,blend_radius_m)
    |   movel(p[0.476957, -0.093528, -0.000100, 0.000000, -3.141593, 0.000000],accel_mss,speed_ms,0,0.000)
    |   movel(p[0.476772, -0.093616, -0.000100, 0.000000, -3.141593, 0.000000],accel_mss,speed_ms,0,0.000)
    |   movel(p[0.476651, -0.093714, -0.000100, 0.000000, -3.141593, 0.000000],accel_mss,speed_ms,0,0.000)
    |   movel(p[0.476536, -0.093828, -0.000100, 0.000000, -3.141593, 0.000000],accel_mss,speed_ms,0,0.000)
    |   movel(p[0.476419, -0.093943, -0.000100, 0.000000, -3.141593, 0.000000],accel_mss,speed_ms,0,0.000)
    |   movel(p[0.476293, -0.094040, -0.000100, 0.000000, -3.141593, 0.000000],accel_mss,speed_ms,0,0.000)
    |   movel(p[0.476175, -0.094108, -0.000100, 0.000000, -3.141593, 0.000000],accel_mss,speed_ms,0,0.000)
    |   movel(p[0.475999, -0.094152, -0.000100, 0.000000, -3.141593, 0.000000],accel_mss,speed_ms,0,0.000)
    |   movel(p[0.475861, -0.094239, -0.000100, 0.000000, -3.141593, 0.000000],accel_mss,speed_ms,0,0.000)
    |   movel(p[0.475709, -0.094360, -0.000100, 0.000000, -3.141593, 0.000000],accel_mss,speed_ms,0,0.000)
    |   movel(p[0.475561, -0.094503, -0.000100, 0.000000, -3.141593, 0.000000],accel_mss,speed_ms,0,0.000)
    |   movel(p[0.475415, -0.094647, -0.000100, 0.000000, -3.141593, 0.000000],accel_mss,speed_ms,0,0.000)
    |   movel(p[0.475269, -0.094768, -0.000100, 0.000000, -3.141593, 0.000000],accel_mss,speed_ms,0,0.000)
    |   movel(p[0.475139, -0.094856, -0.000100, 0.000000, -3.141593, 0.000000],accel_mss,speed_ms,0,0.000)
    |   speed_ms    = 0.050
    |   movel(p[0.475139, -0.094856, 0.003000, 0.000000, -3.141593, 0.000000],accel_mss,speed_ms,0,blend_radius_m)
    |   speed_ms    = 1.000
    |   movel(p[0.475139, -0.094856, 0.015000, 0.000000, -3.141593, 0.000000],accel_mss,speed_ms,0,blend_radius_m)
    |   movel(p[0.452673, -0.050477, 0.015000, 0.000000, -3.141593, 0.000000],accel_mss,speed_ms,0,blend_radius_m)
    |   movel(p[0.452673, -0.050477, 0.003000, 0.000000, -3.141593, 0.000000],accel_mss,speed_ms,0,blend_radius_m)
    |   speed_ms    = 0.050
    |   movel(p[0.452673, -0.050477, -0.000100, 0.000000, -3.141593, 0.000000],accel_mss,speed_ms,0,blend_radius_m)
    |   speed_ms    = 0.083
    |   movel(p[0.452152, -0.050708, -0.000100, 0.000000, -3.141593, 0.000000],accel_mss,speed_ms,0,blend_radius_m)
    |   movel(p[0.451754, -0.050778, -0.000100, 0.000000, 3.141593, 0.000000],accel_mss,speed_ms,0,0.000)
    |   movel(p[0.451576, -0.050755, -0.000100, 0.000000, -3.141593, 0.000000],accel_mss,speed_ms,0,0.000)
    |   movel(p[0.451370, -0.050683, -0.000100, 0.000000, -3.141593, 0.000000],accel_mss,speed_ms,0,0.000)
    |   movel(p[0.451170, -0.050577, -0.000100, 0.000000, 3.141593, 0.000000],accel_mss,speed_ms,0,0.000)
    |   movel(p[0.451008, -0.050452, -0.000100, 0.000000, -3.141593, 0.000000],accel_mss,speed_ms,0,0.000)
    |   movel(p[0.450800, -0.050187, -0.000100, 0.000000, -3.141593, 0.000000],accel_mss,speed_ms,0,0.000)
    |   movel(p[0.450670, -0.049864, -0.000100, 0.000000, 3.141593, 0.000000],accel_mss,speed_ms,0,0.000)
    |   movel(p[0.450690, -0.049683, -0.000100, 0.000000, -3.141593, 0.000000],accel_mss,speed_ms,0,0.000)
    |   movel(p[0.450806, -0.049650, -0.000100, 0.000000, -3.141593, 0.000000],accel_mss,speed_ms,0,0.000)
    |   movel(p[0.450997, -0.049670, -0.000100, 0.000000, -3.141593, 0.000000],accel_mss,speed_ms,0,0.000)
    |   movel(p[0.451508, -0.049463, -0.000100, 0.000000, -3.141593, 0.000000],accel_mss,speed_ms,0,blend_radius_m)
    |   movel(p[0.452133, -0.049158, -0.000100, 0.000000, -3.141593, 0.000000],accel_mss,speed_ms,0,blend_radius_m)
    |   movel(p[0.452836, -0.048755, -0.000100, 0.000000, -3.141593, 0.000000],accel_mss,speed_ms,0,blend_radius_m)
    |   movel(p[0.453403, -0.048472, -0.000100, 0.000000, -3.141593, 0.000000],accel_mss,speed_ms,0,blend_radius_m)
    |   movel(p[0.453863, -0.048387, -0.000100, 0.000000, -3.141593, 0.000000],accel_mss,speed_ms,0,0.000)
    |   movel(p[0.454211, -0.048496, -0.000100, 0.000000, -3.141593, 0.000000],accel_mss,speed_ms,0,0.000)
    |   movel(p[0.454450, -0.048779, -0.000100, 0.000000, -3.141593, 0.000000],accel_mss,speed_ms,0,0.000)
    |   movel(p[0.454538, -0.048991, -0.000100, 0.000000, -3.141593, 0.000000],accel_mss,speed_ms,0,0.000)
    |   movel(p[0.454557, -0.049114, -0.000100, 0.000000, -3.141593, 0.000000],accel_mss,speed_ms,0,0.000)
    |   movel(p[0.454432, -0.049246, -0.000100, 0.000000, -3.141593, 0.000000],accel_mss,speed_ms,0,0.000)
    |   movel(p[0.454326, -0.049297, -0.000100, 0.000000, -3.141593, 0.000000],accel_mss,speed_ms,0,0.000)
    |   movel(p[0.454152, -0.049415, -0.000100, 0.000000, -3.141593, 0.000000],accel_mss,speed_ms,0,0.000)
    |   movel(p[0.453955, -0.049564, -0.000100, 0.000000, -3.141593, 0.000000],accel_mss,speed_ms,0,0.000)
    |   movel(p[0.453759, -0.049728, -0.000100, 0.000000, -3.141593, 0.000000],accel_mss,speed_ms,0,0.000)
    |   movel(p[0.453231, -0.050139, -0.000100, 0.000000, -3.141593, 0.000000],accel_mss,speed_ms,0,blend_radius_m)
    |   movel(p[0.452673, -0.050477, -0.000100, 0.000000, -3.141593, 0.000000],accel_mss,speed_ms,0,blend_radius_m)
    |   speed_ms    = 0.050
    |   movel(p[0.452673, -0.050477, 0.003000, 0.000000, -3.141593, 0.000000],accel_mss,speed_ms,0,blend_radius_m)
    |   speed_ms    = 1.000
    |   movel(p[0.452673, -0.050477, 0.015000, 0.000000, -3.141593, 0.000000],accel_mss,speed_ms,0,blend_radius_m)
    |   movel(p[0.461587, -0.045373, 0.015000, 0.000000, -3.141593, 0.000000],accel_mss,speed_ms,0,blend_radius_m)
    |   movel(p[0.461587, -0.045373, 0.003000, 0.000000, -3.141593, 0.000000],accel_mss,speed_ms,0,blend_radius_m)
    |   speed_ms    = 0.050
    |   movel(p[0.461587, -0.045373, -0.000100, 0.000000, -3.141593, 0.000000],accel_mss,speed_ms,0,blend_radius_m)
    |   speed_ms    = 0.083
    |   movel(p[0.461416, -0.044959, -0.000100, 0.000000, -3.141593, 0.000000],accel_mss,speed_ms,0,0.000)
    |   movel(p[0.461322, -0.044504, -0.000100, 0.000000, -3.141593, 0.000000],accel_mss,speed_ms,0,0.000)
    |   movel(p[0.461317, -0.044135, -0.000100, 0.000000, -3.141593, 0.000000],accel_mss,speed_ms,0,0.000)
    |   movel(p[0.461433, -0.044028, -0.000100, 0.000000, -3.141593, 0.000000],accel_mss,speed_ms,0,0.000)
    |   movel(p[0.461646, -0.044119, -0.000100, 0.000000, 3.141593, 0.000000],accel_mss,speed_ms,0,0.000)
    |   movel(p[0.461986, -0.044507, -0.000100, 0.000000, -3.141593, 0.000000],accel_mss,speed_ms,0,blend_radius_m)
    |   movel(p[0.462303, -0.044962, -0.000100, 0.000000, -3.141593, 0.000000],accel_mss,speed_ms,0,blend_radius_m)
    |   movel(p[0.462493, -0.045369, -0.000100, 0.000000, -3.141593, 0.000000],accel_mss,speed_ms,0,0.000)
    |   movel(p[0.462578, -0.045926, -0.000100, 0.000000, -3.141593, 0.000000],accel_mss,speed_ms,0,blend_radius_m)
    |   movel(p[0.462371, -0.046131, -0.000100, 0.000000, -3.141593, 0.000000],accel_mss,speed_ms,0,0.000)
    |   movel(p[0.461987, -0.045956, -0.000100, 0.000000, 3.141593, 0.000000],accel_mss,speed_ms,0,0.000)
    |   movel(p[0.461587, -0.045373, -0.000100, 0.000000, -3.141593, 0.000000],accel_mss,speed_ms,0,blend_radius_m)
    |   speed_ms    = 0.050
    |   movel(p[0.461587, -0.045373, 0.003000, 0.000000, -3.141593, 0.000000],accel_mss,speed_ms,0,blend_radius_m)
    |   speed_ms    = 1.000
    |   movel(p[0.461587, -0.045373, 0.015000, 0.000000, -3.141593, 0.000000],accel_mss,speed_ms,0,blend_radius_m)
    |   movel(p[0.458150, -0.048329, 0.015000, 0.000000, -3.141593, 0.000000],accel_mss,speed_ms,0,blend_radius_m)
    |   movel(p[0.458150, -0.048329, 0.003000, 0.000000, -3.141593, 0.000000],accel_mss,speed_ms,0,blend_radius_m)
    |   speed_ms    = 0.050
    |   movel(p[0.458150, -0.048329, -0.000100, 0.000000, -3.141593, 0.000000],accel_mss,speed_ms,0,blend_radius_m)
    |   speed_ms    = 0.083
    |   movel(p[0.458072, -0.048891, -0.000100, 0.000000, -3.141593, 0.000000],accel_mss,speed_ms,0,blend_radius_m)
    |   movel(p[0.457923, -0.049563, -0.000100, 0.000000, -3.141593, 0.000000],accel_mss,speed_ms,0,blend_radius_m)
    |   movel(p[0.457708, -0.050253, -0.000100, 0.000000, -3.141593, 0.000000],accel_mss,speed_ms,0,blend_radius_m)
    |   movel(p[0.457599, -0.050573, -0.000100, 0.000000, -3.141593, 0.000000],accel_mss,speed_ms,0,0.000)
    |   movel(p[0.457491, -0.050915, -0.000100, 0.000000, 3.141593, 0.000000],accel_mss,speed_ms,0,0.000)
    |   movel(p[0.457400, -0.051229, -0.000100, 0.000000, -3.141593, 0.000000],accel_mss,speed_ms,0,0.000)
    |   movel(p[0.457345, -0.051453, -0.000100, 0.000000, -3.141593, 0.000000],accel_mss,speed_ms,0,0.000)
    |   movel(p[0.457272, -0.051702, -0.000100, 0.000000, 3.141593, 0.000000],accel_mss,speed_ms,0,0.000)
    |   movel(p[0.457095, -0.052138, -0.000100, 0.000000, 3.141593, 0.000000],accel_mss,speed_ms,0,0.000)
    |   movel(p[0.456873, -0.052641, -0.000100, 0.000000, 3.141593, 0.000000],accel_mss,speed_ms,0,blend_radius_m)
    |   movel(p[0.456628, -0.053152, -0.000100, 0.000000, 3.141593, 0.000000],accel_mss,speed_ms,0,blend_radius_m)
    |   movel(p[0.456240, -0.053863, -0.000100, 0.000000, -3.141593, 0.000000],accel_mss,speed_ms,0,blend_radius_m)
    |   movel(p[0.455859, -0.054418, -0.000100, 0.000000, -3.141593, 0.000000],accel_mss,speed_ms,0,blend_radius_m)
    |   movel(p[0.455364, -0.054980, -0.000100, 0.000000, -3.141593, 0.000000],accel_mss,speed_ms,0,blend_radius_m)
    |   movel(p[0.454592, -0.055740, -0.000100, 0.000000, 3.141593, 0.000000],accel_mss,speed_ms,0,blend_radius_m)
    |   movel(p[0.454039, -0.056253, -0.000100, 0.000000, -3.141593, 0.000000],accel_mss,speed_ms,0,blend_radius_m)
    |   movel(p[0.453551, -0.056685, -0.000100, 0.000000, -3.141593, 0.000000],accel_mss,speed_ms,0,blend_radius_m)
    |   movel(p[0.453128, -0.057045, -0.000100, 0.000000, 3.141593, 0.000000],accel_mss,speed_ms,0,blend_radius_m)
    |   movel(p[0.452947, -0.057093, -0.000100, 0.000000, 3.141593, 0.000000],accel_mss,speed_ms,0,0.000)
    |   movel(p[0.452729, -0.057171, -0.000100, 0.000000, -3.141593, 0.000000],accel_mss,speed_ms,0,0.000)
    |   movel(p[0.452470, -0.057273, -0.000100, 0.000000, -3.141593, 0.000000],accel_mss,speed_ms,0,0.000)
    |   movel(p[0.452190, -0.057394, -0.000100, 0.000000, -3.141593, 0.000000],accel_mss,speed_ms,0,0.000)
    |   movel(p[0.451132, -0.057858, -0.000100, 0.000000, -3.141593, 0.000000],accel_mss,speed_ms,0,blend_radius_m)
    |   movel(p[0.450496, -0.058104, -0.000100, 0.000000, -3.141593, 0.000000],accel_mss,speed_ms,0,blend_radius_m)
    |   movel(p[0.449976, -0.058252, -0.000100, 0.000000, 3.141593, 0.000000],accel_mss,speed_ms,0,blend_radius_m)
    |   movel(p[0.449386, -0.058362, -0.000100, 0.000000, -3.141593, 0.000000],accel_mss,speed_ms,0,blend_radius_m)
    |   movel(p[0.449206, -0.058390, -0.000100, 0.000000, -3.141593, 0.000000],accel_mss,speed_ms,0,0.000)
    |   movel(p[0.448833, -0.058449, -0.000100, 0.000000, -3.141593, 0.000000],accel_mss,speed_ms,0,0.000)
    |   movel(p[0.448391, -0.058521, -0.000100, 0.000000, 3.141593, 0.000000],accel_mss,speed_ms,0,0.000)
    |   movel(p[0.447924, -0.058597, -0.000100, 0.000000, -3.141593, 0.000000],accel_mss,speed_ms,0,0.000)
    |   movel(p[0.447245, -0.058688, -0.000100, 0.000000, -3.141593, 0.000000],accel_mss,speed_ms,0,blend_radius_m)
    |   movel(p[0.446703, -0.058711, -0.000100, 0.000000, 3.141593, 0.000000],accel_mss,speed_ms,0,blend_radius_m)
    |   movel(p[0.446118, -0.058669, -0.000100, 0.000000, -3.141593, 0.000000],accel_mss,speed_ms,0,blend_radius_m)
    |   movel(p[0.445273, -0.058549, -0.000100, 0.000000, -3.141593, 0.000000],accel_mss,speed_ms,0,blend_radius_m)
    |   movel(p[0.444641, -0.058432, -0.000100, 0.000000, -3.141593, 0.000000],accel_mss,speed_ms,0,blend_radius_m)
    |   movel(p[0.444090, -0.058299, -0.000100, 0.000000, -3.141593, 0.000000],accel_mss,speed_ms,0,blend_radius_m)
    |   movel(p[0.443653, -0.058161, -0.000100, 0.000000, 3.141593, 0.000000],accel_mss,speed_ms,0,0.000)
    |   movel(p[0.443412, -0.058031, -0.000100, 0.000000, -3.141593, 0.000000],accel_mss,speed_ms,0,0.000)
    |   movel(p[0.443272, -0.057922, -0.000100, 0.000000, -3.141593, 0.000000],accel_mss,speed_ms,0,0.000)
    |   movel(p[0.443160, -0.057824, -0.000100, 0.000000, -3.141593, 0.000000],accel_mss,speed_ms,0,0.000)
    |   movel(p[0.443077, -0.057741, -0.000100, 0.000000, -3.141593, 0.000000],accel_mss,speed_ms,0,0.000)
    |   movel(p[0.443318, -0.057729, -0.000100, 0.000000, -3.141593, 0.000000],accel_mss,speed_ms,0,0.000)
    |   movel(p[0.443564, -0.057764, -0.000100, 0.000000, -3.141593, 0.000000],accel_mss,speed_ms,0,0.000)
    |   movel(p[0.443849, -0.057814, -0.000100, 0.000000, 3.141593, 0.000000],accel_mss,speed_ms,0,0.000)
    |   movel(p[0.445456, -0.057913, -0.000100, 0.000000, -3.141593, 0.000000],accel_mss,speed_ms,0,blend_radius_m)
    |   movel(p[0.447464, -0.057659, -0.000100, 0.000000, -3.141593, 0.000000],accel_mss,speed_ms,0,blend_radius_m)
    |   movel(p[0.449460, -0.057147, -0.000100, 0.000000, -3.141593, 0.000000],accel_mss,speed_ms,0,blend_radius_m)
    |   movel(p[0.451036, -0.056444, -0.000100, 0.000000, -3.141593, 0.000000],accel_mss,speed_ms,0,blend_radius_m)
    |   movel(p[0.451197, -0.056354, -0.000100, 0.000000, -3.141593, 0.000000],accel_mss,speed_ms,0,0.000)
    |   movel(p[0.451454, -0.056217, -0.000100, 0.000000, -3.141593, 0.000000],accel_mss,speed_ms,0,0.000)
    |   movel(p[0.451746, -0.056065, -0.000100, 0.000000, -3.141593, 0.000000],accel_mss,speed_ms,0,0.000)
    |   movel(p[0.452036, -0.055917, -0.000100, 0.000000, -3.141593, 0.000000],accel_mss,speed_ms,0,0.000)
    |   movel(p[0.452317, -0.055766, -0.000100, 0.000000, -3.141593, 0.000000],accel_mss,speed_ms,0,0.000)
    |   movel(p[0.452584, -0.055604, -0.000100, 0.000000, -3.141593, 0.000000],accel_mss,speed_ms,0,0.000)
    |   movel(p[0.452804, -0.055452, -0.000100, 0.000000, -3.141593, 0.000000],accel_mss,speed_ms,0,0.000)
    |   movel(p[0.452917, -0.055346, -0.000100, 0.000000, -3.141593, 0.000000],accel_mss,speed_ms,0,0.000)
    |   movel(p[0.452999, -0.055263, -0.000100, 0.000000, -3.141593, 0.000000],accel_mss,speed_ms,0,0.000)
    |   movel(p[0.453096, -0.055192, -0.000100, 0.000000, -3.141593, 0.000000],accel_mss,speed_ms,0,0.000)
    |   movel(p[0.453192, -0.055144, -0.000100, 0.000000, 3.141593, 0.000000],accel_mss,speed_ms,0,0.000)
    |   movel(p[0.453506, -0.055035, -0.000100, 0.000000, -3.141593, 0.000000],accel_mss,speed_ms,0,0.000)
    |   movel(p[0.454231, -0.054329, -0.000100, 0.000000, -3.141593, 0.000000],accel_mss,speed_ms,0,blend_radius_m)
    |   movel(p[0.454909, -0.053619, -0.000100, 0.000000, -3.141593, 0.000000],accel_mss,speed_ms,0,blend_radius_m)
    |   movel(p[0.455244, -0.053159, -0.000100, 0.000000, -3.141593, 0.000000],accel_mss,speed_ms,0,blend_radius_m)
    |   movel(p[0.455333, -0.053000, -0.000100, 0.000000, -3.141593, 0.000000],accel_mss,speed_ms,0,0.000)
    |   movel(p[0.455430, -0.052818, -0.000100, 0.000000, -3.141593, 0.000000],accel_mss,speed_ms,0,0.000)
    |   movel(p[0.455520, -0.052640, -0.000100, 0.000000, -3.141593, 0.000000],accel_mss,speed_ms,0,0.000)
    |   movel(p[0.455589, -0.052497, -0.000100, 0.000000, -3.141593, 0.000000],accel_mss,speed_ms,0,0.000)
    |   movel(p[0.455660, -0.052365, -0.000100, 0.000000, -3.141593, 0.000000],accel_mss,speed_ms,0,0.000)
    |   movel(p[0.455759, -0.052222, -0.000100, 0.000000, -3.141593, 0.000000],accel_mss,speed_ms,0,0.000)
    |   movel(p[0.455868, -0.052090, -0.000100, 0.000000, -3.141593, 0.000000],accel_mss,speed_ms,0,0.000)
    |   movel(p[0.455970, -0.051991, -0.000100, 0.000000, -3.141593, 0.000000],accel_mss,speed_ms,0,0.000)
    |   movel(p[0.456062, -0.051895, -0.000100, 0.000000, -3.141593, 0.000000],accel_mss,speed_ms,0,0.000)
    |   movel(p[0.456140, -0.051770, -0.000100, 0.000000, 3.141593, 0.000000],accel_mss,speed_ms,0,0.000)
    |   movel(p[0.456193, -0.051638, -0.000100, 0.000000, 3.141593, 0.000000],accel_mss,speed_ms,0,0.000)
    |   movel(p[0.456211, -0.051519, -0.000100, 0.000000, 3.141593, 0.000000],accel_mss,speed_ms,0,0.000)
    |   movel(p[0.456222, -0.051408, -0.000100, 0.000000, -3.141593, 0.000000],accel_mss,speed_ms,0,0.000)
    |   movel(p[0.456254, -0.051300, -0.000100, 0.000000, -3.141593, 0.000000],accel_mss,speed_ms,0,0.000)
    |   movel(p[0.456301, -0.051210, -0.000100, 0.000000, 3.141593, 0.000000],accel_mss,speed_ms,0,0.000)
    |   movel(p[0.456437, -0.051075, -0.000100, 0.000000, -3.141593, 0.000000],accel_mss,speed_ms,0,0.000)
    |   movel(p[0.456627, -0.050757, -0.000100, 0.000000, -3.141593, 0.000000],accel_mss,speed_ms,0,0.000)
    |   movel(p[0.456842, -0.050369, -0.000100, 0.000000, -3.141593, 0.000000],accel_mss,speed_ms,0,0.000)
    |   movel(p[0.457070, -0.049927, -0.000100, 0.000000, -3.141593, 0.000000],accel_mss,speed_ms,0,0.000)
    |   movel(p[0.457612, -0.048842, -0.000100, 0.000000, -3.141593, 0.000000],accel_mss,speed_ms,0,blend_radius_m)
    |   movel(p[0.457818, -0.048462, -0.000100, 0.000000, -3.141593, 0.000000],accel_mss,speed_ms,0,0.000)
    |   movel(p[0.457947, -0.048280, -0.000100, 0.000000, -3.141593, 0.000000],accel_mss,speed_ms,0,0.000)
    |   movel(p[0.458060, -0.048228, -0.000100, 0.000000, -3.141593, 0.000000],accel_mss,speed_ms,0,0.000)
    |   movel(p[0.458150, -0.048329, -0.000100, 0.000000, -3.141593, 0.000000],accel_mss,speed_ms,0,0.000)
    |   speed_ms    = 0.050
    |   movel(p[0.458150, -0.048329, 0.003000, 0.000000, -3.141593, 0.000000],accel_mss,speed_ms,0,blend_radius_m)
    |   speed_ms    = 1.000
    |   movel(p[0.458150, -0.048329, 0.015000, 0.000000, -3.141593, 0.000000],accel_mss,speed_ms,0,blend_radius_m)
    |   movel(p[0.460013, -0.046384, 0.015000, 0.000000, -3.141593, 0.000000],accel_mss,speed_ms,0,blend_radius_m)
    |   movel(p[0.460013, -0.046384, 0.003000, 0.000000, -3.141593, 0.000000],accel_mss,speed_ms,0,blend_radius_m)
    |   speed_ms    = 0.050
    |   movel(p[0.460013, -0.046384, -0.000100, 0.000000, -3.141593, 0.000000],accel_mss,speed_ms,0,blend_radius_m)
    |   speed_ms    = 0.083
    |   movel(p[0.459961, -0.046278, -0.000100, 0.000000, -3.141593, 0.000000],accel_mss,speed_ms,0,0.000)
    |   movel(p[0.460025, -0.046172, -0.000100, 0.000000, 3.141593, 0.000000],accel_mss,speed_ms,0,0.000)
    |   movel(p[0.460180, -0.046128, -0.000100, 0.000000, -3.141593, 0.000000],accel_mss,speed_ms,0,0.000)
    |   movel(p[0.460462, -0.046184, -0.000100, 0.000000, 3.141593, 0.000000],accel_mss,speed_ms,0,0.000)
    |   movel(p[0.460926, -0.046394, -0.000100, 0.000000, -3.141593, 0.000000],accel_mss,speed_ms,0,blend_radius_m)
    |   movel(p[0.461377, -0.046637, -0.000100, 0.000000, -3.141593, 0.000000],accel_mss,speed_ms,0,blend_radius_m)
    |   movel(p[0.461457, -0.046771, -0.000100, 0.000000, -3.141593, 0.000000],accel_mss,speed_ms,0,0.000)
    |   movel(p[0.461379, -0.046920, -0.000100, 0.000000, -3.141593, 0.000000],accel_mss,speed_ms,0,0.000)
    |   movel(p[0.461177, -0.046976, -0.000100, 0.000000, -3.141593, 0.000000],accel_mss,speed_ms,0,0.000)
    |   movel(p[0.460904, -0.046913, -0.000100, 0.000000, -3.141593, 0.000000],accel_mss,speed_ms,0,0.000)
    |   movel(p[0.460656, -0.046747, -0.000100, 0.000000, 3.141593, 0.000000],accel_mss,speed_ms,0,0.000)
    |   movel(p[0.460513, -0.046625, -0.000100, 0.000000, -3.141593, 0.000000],accel_mss,speed_ms,0,0.000)
    |   movel(p[0.460364, -0.046522, -0.000100, 0.000000, -3.141593, 0.000000],accel_mss,speed_ms,0,0.000)
    |   movel(p[0.460229, -0.046449, -0.000100, 0.000000, -3.141593, 0.000000],accel_mss,speed_ms,0,0.000)
    |   movel(p[0.460071, -0.046417, -0.000100, 0.000000, -3.141593, 0.000000],accel_mss,speed_ms,0,0.000)
    |   speed_ms    = 0.050
    |   movel(p[0.460013, -0.046384, 0.003000, 0.000000, -3.141593, 0.000000],accel_mss,speed_ms,0,blend_radius_m)
    |   speed_ms    = 1.000
    |   movel(p[0.460013, -0.046384, 0.015000, 0.000000, -3.141593, 0.000000],accel_mss,speed_ms,0,blend_radius_m)
    |   movel(p[0.460275, -0.045372, 0.015000, 0.000000, -3.141593, 0.000000],accel_mss,speed_ms,0,blend_radius_m)
    |   movel(p[0.460275, -0.045372, 0.003000, 0.000000, -3.141593, 0.000000],accel_mss,speed_ms,0,blend_radius_m)
    |   speed_ms    = 0.050
    |   movel(p[0.460275, -0.045372, -0.000100, 0.000000, -3.141593, 0.000000],accel_mss,speed_ms,0,blend_radius_m)
    |   speed_ms    = 0.083
    |   movel(p[0.459823, -0.045339, -0.000100, 0.000000, 3.141593, 0.000000],accel_mss,speed_ms,0,0.000)
    |   movel(p[0.459426, -0.045318, -0.000100, 0.000000, -3.141593, 0.000000],accel_mss,speed_ms,0,0.000)
    |   movel(p[0.459076, -0.045329, -0.000100, 0.000000, 3.141593, 0.000000],accel_mss,speed_ms,0,0.000)
    |   movel(p[0.458787, -0.045370, -0.000100, 0.000000, -3.141593, 0.000000],accel_mss,speed_ms,0,0.000)
    |   movel(p[0.458582, -0.045442, -0.000100, 0.000000, -3.141593, 0.000000],accel_mss,speed_ms,0,0.000)
    |   movel(p[0.458309, -0.045545, -0.000100, 0.000000, -3.141593, 0.000000],accel_mss,speed_ms,0,0.000)
    |   movel(p[0.458061, -0.045557, -0.000100, 0.000000, -3.141593, 0.000000],accel_mss,speed_ms,0,0.000)
    |   movel(p[0.457819, -0.045476, -0.000100, 0.000000, -3.141593, 0.000000],accel_mss,speed_ms,0,0.000)
    |   movel(p[0.457561, -0.045298, -0.000100, 0.000000, -3.141593, 0.000000],accel_mss,speed_ms,0,0.000)
    |   movel(p[0.457413, -0.045191, -0.000100, 0.000000, -3.141593, 0.000000],accel_mss,speed_ms,0,0.000)
    |   movel(p[0.457055, -0.044980, -0.000100, 0.000000, 3.141593, 0.000000],accel_mss,speed_ms,0,0.000)
    |   movel(p[0.456624, -0.044738, -0.000100, 0.000000, -3.141593, 0.000000],accel_mss,speed_ms,0,0.000)
    |   movel(p[0.456156, -0.044487, -0.000100, 0.000000, -3.141593, 0.000000],accel_mss,speed_ms,0,blend_radius_m)
    |   movel(p[0.454347, -0.043738, -0.000100, 0.000000, -3.141593, 0.000000],accel_mss,speed_ms,0,blend_radius_m)
    |   movel(p[0.452107, -0.043177, -0.000100, 0.000000, 3.141593, 0.000000],accel_mss,speed_ms,0,blend_radius_m)
    |   movel(p[0.449872, -0.042876, -0.000100, 0.000000, -3.141593, 0.000000],accel_mss,speed_ms,0,blend_radius_m)
    |   movel(p[0.448094, -0.042938, -0.000100, 0.000000, -3.141593, 0.000000],accel_mss,speed_ms,0,blend_radius_m)
    |   movel(p[0.446696, -0.043209, -0.000100, 0.000000, -3.141593, 0.000000],accel_mss,speed_ms,0,blend_radius_m)
    |   movel(p[0.445440, -0.043586, -0.000100, 0.000000, 3.141593, 0.000000],accel_mss,speed_ms,0,blend_radius_m)
    |   movel(p[0.444430, -0.044025, -0.000100, 0.000000, -3.141593, 0.000000],accel_mss,speed_ms,0,blend_radius_m)
    |   movel(p[0.443832, -0.044484, -0.000100, 0.000000, -3.141593, 0.000000],accel_mss,speed_ms,0,blend_radius_m)
    |   movel(p[0.443694, -0.044619, -0.000100, 0.000000, -3.141593, 0.000000],accel_mss,speed_ms,0,0.000)
    |   movel(p[0.443523, -0.044754, -0.000100, 0.000000, -3.141593, 0.000000],accel_mss,speed_ms,0,0.000)
    |   movel(p[0.443347, -0.044870, -0.000100, 0.000000, -3.141593, 0.000000],accel_mss,speed_ms,0,0.000)
    |   movel(p[0.443196, -0.044943, -0.000100, 0.000000, -3.141593, 0.000000],accel_mss,speed_ms,0,0.000)
    |   movel(p[0.443056, -0.045018, -0.000100, 0.000000, -3.141593, 0.000000],accel_mss,speed_ms,0,0.000)
    |   movel(p[0.442917, -0.045135, -0.000100, 0.000000, -3.141593, 0.000000],accel_mss,speed_ms,0,0.000)
    |   movel(p[0.442800, -0.045273, -0.000100, 0.000000, -3.141593, 0.000000],accel_mss,speed_ms,0,0.000)
    |   movel(p[0.442725, -0.045413, -0.000100, 0.000000, -3.141593, 0.000000],accel_mss,speed_ms,0,0.000)
    |   movel(p[0.442652, -0.045565, -0.000100, 0.000000, -3.141593, 0.000000],accel_mss,speed_ms,0,0.000)
    |   movel(p[0.442537, -0.045740, -0.000100, 0.000000, -3.141593, 0.000000],accel_mss,speed_ms,0,0.000)
    |   movel(p[0.442402, -0.045911, -0.000100, 0.000000, -3.141593, 0.000000],accel_mss,speed_ms,0,0.000)
    |   movel(p[0.442267, -0.046050, -0.000100, 0.000000, -3.141593, 0.000000],accel_mss,speed_ms,0,0.000)
    |   movel(p[0.442029, -0.046325, -0.000100, 0.000000, 3.141593, 0.000000],accel_mss,speed_ms,0,0.000)
    |   movel(p[0.441763, -0.046766, -0.000100, 0.000000, -3.141593, 0.000000],accel_mss,speed_ms,0,blend_radius_m)
    |   movel(p[0.441487, -0.047332, -0.000100, 0.000000, -3.141593, 0.000000],accel_mss,speed_ms,0,blend_radius_m)
    |   movel(p[0.441211, -0.048003, -0.000100, 0.000000, -3.141593, 0.000000],accel_mss,speed_ms,0,blend_radius_m)
    |   movel(p[0.441009, -0.048282, -0.000100, 0.000000, 3.141593, 0.000000],accel_mss,speed_ms,0,0.000)
    |   movel(p[0.440736, -0.048344, -0.000100, 0.000000, 3.141593, 0.000000],accel_mss,speed_ms,0,0.000)
    |   movel(p[0.440366, -0.048161, -0.000100, 0.000000, -3.141593, 0.000000],accel_mss,speed_ms,0,0.000)
    |   movel(p[0.439855, -0.047690, -0.000100, 0.000000, -3.141593, 0.000000],accel_mss,speed_ms,0,blend_radius_m)
    |   movel(p[0.439577, -0.047416, -0.000100, 0.000000, -3.141593, 0.000000],accel_mss,speed_ms,0,0.000)
    |   movel(p[0.439294, -0.047162, -0.000100, 0.000000, -3.141593, 0.000000],accel_mss,speed_ms,0,0.000)
    |   movel(p[0.439043, -0.046958, -0.000100, 0.000000, -3.141593, 0.000000],accel_mss,speed_ms,0,0.000)
    |   movel(p[0.438886, -0.046862, -0.000100, 0.000000, -3.141593, 0.000000],accel_mss,speed_ms,0,0.000)
    |   movel(p[0.438740, -0.046789, -0.000100, 0.000000, 3.141593, 0.000000],accel_mss,speed_ms,0,0.000)
    |   movel(p[0.438542, -0.046678, -0.000100, 0.000000, -3.141593, 0.000000],accel_mss,speed_ms,0,0.000)
    |   movel(p[0.438330, -0.046551, -0.000100, 0.000000, -3.141593, 0.000000],accel_mss,speed_ms,0,0.000)
    |   movel(p[0.438136, -0.046428, -0.000100, 0.000000, -3.141593, 0.000000],accel_mss,speed_ms,0,0.000)
    |   movel(p[0.437421, -0.046004, -0.000100, 0.000000, -3.141593, 0.000000],accel_mss,speed_ms,0,blend_radius_m)
    |   movel(p[0.436390, -0.045479, -0.000100, 0.000000, -3.141593, 0.000000],accel_mss,speed_ms,0,blend_radius_m)
    |   movel(p[0.435364, -0.044995, -0.000100, 0.000000, -3.141593, 0.000000],accel_mss,speed_ms,0,blend_radius_m)
    |   movel(p[0.434919, -0.044861, -0.000100, 0.000000, 3.141593, 0.000000],accel_mss,speed_ms,0,0.000)
    |   movel(p[0.433354, -0.044623, -0.000100, 0.000000, -3.141593, 0.000000],accel_mss,speed_ms,0,blend_radius_m)
    |   movel(p[0.432422, -0.044522, -0.000100, 0.000000, 3.141593, 0.000000],accel_mss,speed_ms,0,blend_radius_m)
    |   movel(p[0.431635, -0.044500, -0.000100, 0.000000, -3.141593, 0.000000],accel_mss,speed_ms,0,blend_radius_m)
    |   movel(p[0.430668, -0.044543, -0.000100, 0.000000, -3.141593, 0.000000],accel_mss,speed_ms,0,blend_radius_m)
    |   movel(p[0.430059, -0.044587, -0.000100, 0.000000, -3.141593, 0.000000],accel_mss,speed_ms,0,blend_radius_m)
    |   movel(p[0.429498, -0.044631, -0.000100, 0.000000, -3.141593, 0.000000],accel_mss,speed_ms,0,blend_radius_m)
    |   movel(p[0.429027, -0.044670, -0.000100, 0.000000, -3.141593, 0.000000],accel_mss,speed_ms,0,0.000)
    |   movel(p[0.428836, -0.044691, -0.000100, 0.000000, -3.141593, 0.000000],accel_mss,speed_ms,0,0.000)
    |   movel(p[0.427123, -0.045042, -0.000100, 0.000000, -3.141593, 0.000000],accel_mss,speed_ms,0,blend_radius_m)
    |   movel(p[0.425657, -0.045602, -0.000100, 0.000000, -3.141593, 0.000000],accel_mss,speed_ms,0,blend_radius_m)
    |   movel(p[0.424330, -0.046426, -0.000100, 0.000000, -3.141593, 0.000000],accel_mss,speed_ms,0,blend_radius_m)
    |   movel(p[0.423032, -0.047566, -0.000100, 0.000000, -3.141593, 0.000000],accel_mss,speed_ms,0,blend_radius_m)
    |   movel(p[0.422546, -0.048049, -0.000100, 0.000000, -3.141593, 0.000000],accel_mss,speed_ms,0,blend_radius_m)
    |   movel(p[0.422119, -0.048457, -0.000100, 0.000000, 3.141593, 0.000000],accel_mss,speed_ms,0,blend_radius_m)
    |   movel(p[0.421747, -0.048799, -0.000100, 0.000000, -3.141593, 0.000000],accel_mss,speed_ms,0,blend_radius_m)
    |   movel(p[0.421587, -0.048770, -0.000100, 0.000000, -3.141593, 0.000000],accel_mss,speed_ms,0,0.000)
    |   movel(p[0.421592, -0.048648, -0.000100, 0.000000, -3.141593, 0.000000],accel_mss,speed_ms,0,0.000)
    |   movel(p[0.421735, -0.048438, -0.000100, 0.000000, -3.141593, 0.000000],accel_mss,speed_ms,0,0.000)
    |   movel(p[0.422011, -0.048153, -0.000100, 0.000000, -3.141593, 0.000000],accel_mss,speed_ms,0,0.000)
    |   movel(p[0.422183, -0.047978, -0.000100, 0.000000, -3.141593, 0.000000],accel_mss,speed_ms,0,0.000)
    |   movel(p[0.422329, -0.047806, -0.000100, 0.000000, 3.141593, 0.000000],accel_mss,speed_ms,0,0.000)
    |   movel(p[0.422437, -0.047656, -0.000100, 0.000000, -3.141593, 0.000000],accel_mss,speed_ms,0,0.000)
    |   movel(p[0.422586, -0.047251, -0.000100, 0.000000, -3.141593, 0.000000],accel_mss,speed_ms,0,0.000)
    |   movel(p[0.424352, -0.045326, -0.000100, 0.000000, -3.141593, 0.000000],accel_mss,speed_ms,0,blend_radius_m)
    |   movel(p[0.426139, -0.043405, -0.000100, 0.000000, -3.141593, 0.000000],accel_mss,speed_ms,0,blend_radius_m)
    |   movel(p[0.426430, -0.043278, -0.000100, 0.000000, -3.141593, 0.000000],accel_mss,speed_ms,0,0.000)
    |   movel(p[0.426529, -0.043245, -0.000100, 0.000000, -3.141593, 0.000000],accel_mss,speed_ms,0,0.000)
    |   movel(p[0.426765, -0.043058, -0.000100, 0.000000, -3.141593, 0.000000],accel_mss,speed_ms,0,0.000)
    |   movel(p[0.427041, -0.042816, -0.000100, 0.000000, 3.141593, 0.000000],accel_mss,speed_ms,0,0.000)
    |   movel(p[0.427336, -0.042528, -0.000100, 0.000000, 3.141593, 0.000000],accel_mss,speed_ms,0,0.000)
    |   movel(p[0.427629, -0.042241, -0.000100, 0.000000, 3.141593, 0.000000],accel_mss,speed_ms,0,0.000)
    |   movel(p[0.427897, -0.041999, -0.000100, 0.000000, -3.141593, 0.000000],accel_mss,speed_ms,0,0.000)
    |   movel(p[0.428128, -0.041807, -0.000100, 0.000000, -3.141593, 0.000000],accel_mss,speed_ms,0,0.000)
    |   movel(p[0.428295, -0.041752, -0.000100, 0.000000, 3.141593, 0.000000],accel_mss,speed_ms,0,0.000)
    |   movel(p[0.428554, -0.041566, -0.000100, 0.000000, -3.141593, 0.000000],accel_mss,speed_ms,0,0.000)
    |   movel(p[0.428857, -0.041333, -0.000100, 0.000000, -3.141593, 0.000000],accel_mss,speed_ms,0,0.000)
    |   movel(p[0.429191, -0.041056, -0.000100, 0.000000, -3.141593, 0.000000],accel_mss,speed_ms,0,0.000)
    |   movel(p[0.429555, -0.040761, -0.000100, 0.000000, -3.141593, 0.000000],accel_mss,speed_ms,0,0.000)
    |   movel(p[0.429951, -0.040471, -0.000100, 0.000000, -3.141593, 0.000000],accel_mss,speed_ms,0,0.000)
    |   movel(p[0.430321, -0.040225, -0.000100, 0.000000, -3.141593, 0.000000],accel_mss,speed_ms,0,0.000)
    |   movel(p[0.430592, -0.040077, -0.000100, 0.000000, -3.141593, 0.000000],accel_mss,speed_ms,0,0.000)
    |   movel(p[0.430811, -0.039969, -0.000100, 0.000000, -3.141593, 0.000000],accel_mss,speed_ms,0,0.000)
    |   movel(p[0.431010, -0.039856, -0.000100, 0.000000, 3.141593, 0.000000],accel_mss,speed_ms,0,0.000)
    |   movel(p[0.431169, -0.039751, -0.000100, 0.000000, 3.141593, 0.000000],accel_mss,speed_ms,0,0.000)
    |   movel(p[0.431290, -0.039618, -0.000100, 0.000000, -3.141593, 0.000000],accel_mss,speed_ms,0,0.000)
    |   movel(p[0.431412, -0.039525, -0.000100, 0.000000, 3.141593, 0.000000],accel_mss,speed_ms,0,0.000)
    |   movel(p[0.431563, -0.039425, -0.000100, 0.000000, -3.141593, 0.000000],accel_mss,speed_ms,0,0.000)
    |   movel(p[0.431726, -0.039333, -0.000100, 0.000000, -3.141593, 0.000000],accel_mss,speed_ms,0,0.000)
    |   movel(p[0.431960, -0.039211, -0.000100, 0.000000, -3.141593, 0.000000],accel_mss,speed_ms,0,0.000)
    |   movel(p[0.432390, -0.038985, -0.000100, 0.000000, -3.141593, 0.000000],accel_mss,speed_ms,0,0.000)
    |   movel(p[0.432893, -0.038720, -0.000100, 0.000000, -3.141593, 0.000000],accel_mss,speed_ms,0,blend_radius_m)
    |   movel(p[0.433412, -0.038448, -0.000100, 0.000000, 3.141593, 0.000000],accel_mss,speed_ms,0,blend_radius_m)
    |   movel(p[0.433944, -0.038176, -0.000100, 0.000000, -3.141593, 0.000000],accel_mss,speed_ms,0,blend_radius_m)
    |   movel(p[0.434489, -0.037916, -0.000100, 0.000000, -3.141593, 0.000000],accel_mss,speed_ms,0,blend_radius_m)
    |   movel(p[0.434973, -0.037700, -0.000100, 0.000000, 3.141593, 0.000000],accel_mss,speed_ms,0,blend_radius_m)
    |   movel(p[0.435287, -0.037583, -0.000100, 0.000000, -3.141593, 0.000000],accel_mss,speed_ms,0,0.000)
    |   movel(p[0.435527, -0.037500, -0.000100, 0.000000, -3.141593, 0.000000],accel_mss,speed_ms,0,0.000)
    |   movel(p[0.435754, -0.037414, -0.000100, 0.000000, -3.141593, 0.000000],accel_mss,speed_ms,0,0.000)
    |   movel(p[0.435943, -0.037333, -0.000100, 0.000000, -3.141593, 0.000000],accel_mss,speed_ms,0,0.000)
    |   movel(p[0.436036, -0.037279, -0.000100, 0.000000, 3.141593, 0.000000],accel_mss,speed_ms,0,0.000)
    |   movel(p[0.436379, -0.037098, -0.000100, 0.000000, -3.141593, 0.000000],accel_mss,speed_ms,0,0.000)
    |   movel(p[0.437384, -0.036765, -0.000100, 0.000000, 3.141593, 0.000000],accel_mss,speed_ms,0,blend_radius_m)
    |   movel(p[0.438577, -0.036405, -0.000100, 0.000000, -3.141593, 0.000000],accel_mss,speed_ms,0,blend_radius_m)
    |   movel(p[0.439861, -0.036058, -0.000100, 0.000000, 3.141593, 0.000000],accel_mss,speed_ms,0,blend_radius_m)
    |   movel(p[0.443288, -0.035424, -0.000100, 0.000000, -3.141593, 0.000000],accel_mss,speed_ms,0,blend_radius_m)
    |   movel(p[0.447124, -0.035178, -0.000100, 0.000000, -3.141593, 0.000000],accel_mss,speed_ms,0,blend_radius_m)
    |   movel(p[0.451004, -0.035322, -0.000100, 0.000000, -3.141593, 0.000000],accel_mss,speed_ms,0,blend_radius_m)
    |   movel(p[0.454561, -0.035863, -0.000100, 0.000000, -3.141593, 0.000000],accel_mss,speed_ms,0,blend_radius_m)
    |   movel(p[0.456004, -0.036199, -0.000100, 0.000000, -3.141593, 0.000000],accel_mss,speed_ms,0,blend_radius_m)
    |   movel(p[0.457480, -0.036584, -0.000100, 0.000000, -3.141593, 0.000000],accel_mss,speed_ms,0,blend_radius_m)
    |   movel(p[0.458827, -0.036962, -0.000100, 0.000000, -3.141593, 0.000000],accel_mss,speed_ms,0,blend_radius_m)
    |   movel(p[0.459132, -0.037118, -0.000100, 0.000000, -3.141593, 0.000000],accel_mss,speed_ms,0,0.000)
    |   movel(p[0.459227, -0.037176, -0.000100, 0.000000, -3.141593, 0.000000],accel_mss,speed_ms,0,0.000)
    |   movel(p[0.459417, -0.037260, -0.000100, 0.000000, -3.141593, 0.000000],accel_mss,speed_ms,0,0.000)
    |   movel(p[0.459645, -0.037348, -0.000100, 0.000000, -3.141593, 0.000000],accel_mss,speed_ms,0,0.000)
    |   movel(p[0.459886, -0.037430, -0.000100, 0.000000, -3.141593, 0.000000],accel_mss,speed_ms,0,0.000)
    |   movel(p[0.460780, -0.037778, -0.000100, 0.000000, -3.141593, 0.000000],accel_mss,speed_ms,0,blend_radius_m)
    |   movel(p[0.462551, -0.038624, -0.000100, 0.000000, 3.141593, 0.000000],accel_mss,speed_ms,0,blend_radius_m)
    |   movel(p[0.464319, -0.039507, -0.000100, 0.000000, -3.141593, 0.000000],accel_mss,speed_ms,0,blend_radius_m)
    |   movel(p[0.465000, -0.039931, -0.000100, 0.000000, 3.141593, 0.000000],accel_mss,speed_ms,0,blend_radius_m)
    |   movel(p[0.465189, -0.040064, -0.000100, 0.000000, 3.141593, 0.000000],accel_mss,speed_ms,0,0.000)
    |   movel(p[0.465372, -0.040176, -0.000100, 0.000000, -3.141593, 0.000000],accel_mss,speed_ms,0,0.000)
    |   movel(p[0.465530, -0.040259, -0.000100, 0.000000, -3.141593, 0.000000],accel_mss,speed_ms,0,0.000)
    |   movel(p[0.465690, -0.040298, -0.000100, 0.000000, -3.141593, 0.000000],accel_mss,speed_ms,0,0.000)
    |   movel(p[0.465800, -0.040366, -0.000100, 0.000000, -3.141593, 0.000000],accel_mss,speed_ms,0,0.000)
    |   movel(p[0.465921, -0.040464, -0.000100, 0.000000, -3.141593, 0.000000],accel_mss,speed_ms,0,0.000)
    |   movel(p[0.466036, -0.040578, -0.000100, 0.000000, -3.141593, 0.000000],accel_mss,speed_ms,0,0.000)
    |   movel(p[0.466153, -0.040693, -0.000100, 0.000000, -3.141593, 0.000000],accel_mss,speed_ms,0,0.000)
    |   movel(p[0.466279, -0.040790, -0.000100, 0.000000, -3.141593, 0.000000],accel_mss,speed_ms,0,0.000)
    |   movel(p[0.466397, -0.040858, -0.000100, 0.000000, -3.141593, 0.000000],accel_mss,speed_ms,0,0.000)
    |   movel(p[0.466573, -0.040902, -0.000100, 0.000000, -3.141593, 0.000000],accel_mss,speed_ms,0,0.000)
    |   movel(p[0.466711, -0.040989, -0.000100, 0.000000, 3.141593, 0.000000],accel_mss,speed_ms,0,0.000)
    |   movel(p[0.466863, -0.041110, -0.000100, 0.000000, -3.141593, 0.000000],accel_mss,speed_ms,0,0.000)
    |   movel(p[0.467011, -0.041253, -0.000100, 0.000000, -3.141593, 0.000000],accel_mss,speed_ms,0,0.000)
    |   movel(p[0.467161, -0.041397, -0.000100, 0.000000, -3.141593, 0.000000],accel_mss,speed_ms,0,0.000)
    |   movel(p[0.467321, -0.041518, -0.000100, 0.000000, -3.141593, 0.000000],accel_mss,speed_ms,0,0.000)
    |   movel(p[0.467468, -0.041604, -0.000100, 0.000000, -3.141593, 0.000000],accel_mss,speed_ms,0,0.000)
    |   movel(p[0.467571, -0.041628, -0.000100, 0.000000, -3.141593, 0.000000],accel_mss,speed_ms,0,0.000)
    |   movel(p[0.467900, -0.041764, -0.000100, 0.000000, -3.141593, 0.000000],accel_mss,speed_ms,0,0.000)
    |   movel(p[0.470169, -0.044022, -0.000100, 0.000000, 3.141593, 0.000000],accel_mss,speed_ms,0,blend_radius_m)
    |   movel(p[0.472426, -0.046292, -0.000100, 0.000000, -3.141593, 0.000000],accel_mss,speed_ms,0,blend_radius_m)
    |   movel(p[0.472561, -0.046621, -0.000100, 0.000000, -3.141593, 0.000000],accel_mss,speed_ms,0,0.000)
    |   movel(p[0.472581, -0.046720, -0.000100, 0.000000, -3.141593, 0.000000],accel_mss,speed_ms,0,0.000)
    |   movel(p[0.472647, -0.046847, -0.000100, 0.000000, 3.141593, 0.000000],accel_mss,speed_ms,0,0.000)
    |   movel(p[0.472741, -0.046979, -0.000100, 0.000000, -3.141593, 0.000000],accel_mss,speed_ms,0,0.000)
    |   movel(p[0.472852, -0.047096, -0.000100, 0.000000, -3.141593, 0.000000],accel_mss,speed_ms,0,0.000)
    |   movel(p[0.472971, -0.047228, -0.000100, 0.000000, 3.141593, 0.000000],accel_mss,speed_ms,0,0.000)
    |   movel(p[0.473086, -0.047409, -0.000100, 0.000000, -3.141593, 0.000000],accel_mss,speed_ms,0,0.000)
    |   movel(p[0.473181, -0.047607, -0.000100, 0.000000, -3.141593, 0.000000],accel_mss,speed_ms,0,0.000)
    |   movel(p[0.473239, -0.047792, -0.000100, 0.000000, -3.141593, 0.000000],accel_mss,speed_ms,0,0.000)
    |   movel(p[0.473286, -0.047964, -0.000100, 0.000000, -3.141593, 0.000000],accel_mss,speed_ms,0,0.000)
    |   movel(p[0.473349, -0.048124, -0.000100, 0.000000, -3.141593, 0.000000],accel_mss,speed_ms,0,0.000)
    |   movel(p[0.473418, -0.048253, -0.000100, 0.000000, 3.141593, 0.000000],accel_mss,speed_ms,0,0.000)
    |   movel(p[0.473739, -0.048610, -0.000100, 0.000000, -3.141593, 0.000000],accel_mss,speed_ms,0,0.000)
    |   movel(p[0.474354, -0.050018, -0.000100, 0.000000, 3.141593, 0.000000],accel_mss,speed_ms,0,blend_radius_m)
    |   movel(p[0.474963, -0.051540, -0.000100, 0.000000, -3.141593, 0.000000],accel_mss,speed_ms,0,blend_radius_m)
    |   movel(p[0.475450, -0.052953, -0.000100, 0.000000, -3.141593, 0.000000],accel_mss,speed_ms,0,blend_radius_m)
    |   movel(p[0.475793, -0.054128, -0.000100, 0.000000, -3.141593, 0.000000],accel_mss,speed_ms,0,blend_radius_m)
    |   movel(p[0.476181, -0.055614, -0.000100, 0.000000, -3.141593, 0.000000],accel_mss,speed_ms,0,blend_radius_m)
    |   movel(p[0.476524, -0.057034, -0.000100, 0.000000, -3.141593, 0.000000],accel_mss,speed_ms,0,blend_radius_m)
    |   movel(p[0.476670, -0.057828, -0.000100, 0.000000, -3.141593, 0.000000],accel_mss,speed_ms,0,blend_radius_m)
    |   movel(p[0.476705, -0.058114, -0.000100, 0.000000, -3.141593, 0.000000],accel_mss,speed_ms,0,0.000)
    |   movel(p[0.476753, -0.058585, -0.000100, 0.000000, -3.141593, 0.000000],accel_mss,speed_ms,0,0.000)
    |   movel(p[0.476802, -0.059125, -0.000100, 0.000000, 3.141593, 0.000000],accel_mss,speed_ms,0,blend_radius_m)
    |   movel(p[0.476848, -0.059666, -0.000100, 0.000000, -3.141593, 0.000000],accel_mss,speed_ms,0,blend_radius_m)
    |   movel(p[0.476900, -0.060322, -0.000100, 0.000000, -3.141593, 0.000000],accel_mss,speed_ms,0,blend_radius_m)
    |   movel(p[0.476952, -0.060978, -0.000100, 0.000000, -3.141593, 0.000000],accel_mss,speed_ms,0,blend_radius_m)
    |   movel(p[0.476577, -0.060978, -0.000100, 0.000000, -3.141593, 0.000000],accel_mss,speed_ms,0,0.000)
    |   movel(p[0.476201, -0.060978, -0.000100, 0.000000, -3.141593, 0.000000],accel_mss,speed_ms,0,0.000)
    |   movel(p[0.475352, -0.061030, -0.000100, 0.000000, -3.141593, 0.000000],accel_mss,speed_ms,0,blend_radius_m)
    |   movel(p[0.474198, -0.061201, -0.000100, 0.000000, -3.141593, 0.000000],accel_mss,speed_ms,0,blend_radius_m)
    |   movel(p[0.473058, -0.061427, -0.000100, 0.000000, -3.141593, 0.000000],accel_mss,speed_ms,0,blend_radius_m)
    |   movel(p[0.472256, -0.061661, -0.000100, 0.000000, -3.141593, 0.000000],accel_mss,speed_ms,0,blend_radius_m)
    |   movel(p[0.471987, -0.061757, -0.000100, 0.000000, -3.141593, 0.000000],accel_mss,speed_ms,0,0.000)
    |   movel(p[0.471732, -0.061842, -0.000100, 0.000000, -3.141593, 0.000000],accel_mss,speed_ms,0,0.000)
    |   movel(p[0.471517, -0.061910, -0.000100, 0.000000, -3.141593, 0.000000],accel_mss,speed_ms,0,0.000)
    |   movel(p[0.471414, -0.061935, -0.000100, 0.000000, -3.141593, 0.000000],accel_mss,speed_ms,0,0.000)
    |   movel(p[0.471232, -0.062007, -0.000100, 0.000000, -3.141593, 0.000000],accel_mss,speed_ms,0,0.000)
    |   movel(p[0.471128, -0.062068, -0.000100, 0.000000, -3.141593, 0.000000],accel_mss,speed_ms,0,0.000)
    |   movel(p[0.471038, -0.062135, -0.000100, 0.000000, -3.141593, 0.000000],accel_mss,speed_ms,0,0.000)
    |   movel(p[0.470933, -0.062207, -0.000100, 0.000000, -3.141593, 0.000000],accel_mss,speed_ms,0,0.000)
    |   movel(p[0.470782, -0.062283, -0.000100, 0.000000, -3.141593, 0.000000],accel_mss,speed_ms,0,0.000)
    |   movel(p[0.470614, -0.062351, -0.000100, 0.000000, -3.141593, 0.000000],accel_mss,speed_ms,0,0.000)
    |   movel(p[0.470453, -0.062400, -0.000100, 0.000000, 3.141593, 0.000000],accel_mss,speed_ms,0,0.000)
    |   movel(p[0.469979, -0.062619, -0.000100, 0.000000, -3.141593, 0.000000],accel_mss,speed_ms,0,blend_radius_m)
    |   movel(p[0.469355, -0.063119, -0.000100, 0.000000, -3.141593, 0.000000],accel_mss,speed_ms,0,blend_radius_m)
    |   movel(p[0.468779, -0.063699, -0.000100, 0.000000, -3.141593, 0.000000],accel_mss,speed_ms,0,blend_radius_m)
    |   movel(p[0.468448, -0.064198, -0.000100, 0.000000, -3.141593, 0.000000],accel_mss,speed_ms,0,blend_radius_m)
    |   movel(p[0.468236, -0.064591, -0.000100, 0.000000, -3.141593, 0.000000],accel_mss,speed_ms,0,0.000)
    |   movel(p[0.468073, -0.064698, -0.000100, 0.000000, -3.141593, 0.000000],accel_mss,speed_ms,0,0.000)
    |   movel(p[0.467895, -0.064637, -0.000100, 0.000000, -3.141593, 0.000000],accel_mss,speed_ms,0,0.000)
    |   movel(p[0.467618, -0.064316, -0.000100, 0.000000, -3.141593, 0.000000],accel_mss,speed_ms,0,0.000)
    |   movel(p[0.467209, -0.063820, -0.000100, 0.000000, -3.141593, 0.000000],accel_mss,speed_ms,0,blend_radius_m)
    |   movel(p[0.466671, -0.063243, -0.000100, 0.000000, -3.141593, 0.000000],accel_mss,speed_ms,0,blend_radius_m)
    |   movel(p[0.466121, -0.062688, -0.000100, 0.000000, 3.141593, 0.000000],accel_mss,speed_ms,0,blend_radius_m)
    |   movel(p[0.465975, -0.062628, -0.000100, 0.000000, -3.141593, 0.000000],accel_mss,speed_ms,0,0.000)
    |   movel(p[0.465794, -0.062520, -0.000100, 0.000000, -3.141593, 0.000000],accel_mss,speed_ms,0,0.000)
    |   movel(p[0.465658, -0.062401, -0.000100, 0.000000, -3.141593, 0.000000],accel_mss,speed_ms,0,0.000)
    |   movel(p[0.465517, -0.062260, -0.000100, 0.000000, -3.141593, 0.000000],accel_mss,speed_ms,0,0.000)
    |   movel(p[0.465378, -0.062121, -0.000100, 0.000000, 3.141593, 0.000000],accel_mss,speed_ms,0,0.000)
    |   movel(p[0.465246, -0.062007, -0.000100, 0.000000, -3.141593, 0.000000],accel_mss,speed_ms,0,0.000)
    |   movel(p[0.465132, -0.061924, -0.000100, 0.000000, -3.141593, 0.000000],accel_mss,speed_ms,0,0.000)
    |   movel(p[0.465016, -0.061911, -0.000100, 0.000000, -3.141593, 0.000000],accel_mss,speed_ms,0,0.000)
    |   movel(p[0.464806, -0.061834, -0.000100, 0.000000, 3.141593, 0.000000],accel_mss,speed_ms,0,0.000)
    |   movel(p[0.464558, -0.061732, -0.000100, 0.000000, -3.141593, 0.000000],accel_mss,speed_ms,0,0.000)
    |   movel(p[0.464282, -0.061608, -0.000100, 0.000000, -3.141593, 0.000000],accel_mss,speed_ms,0,0.000)
    |   movel(p[0.463998, -0.061482, -0.000100, 0.000000, 3.141593, 0.000000],accel_mss,speed_ms,0,0.000)
    |   movel(p[0.463727, -0.061375, -0.000100, 0.000000, -3.141593, 0.000000],accel_mss,speed_ms,0,0.000)
    |   movel(p[0.463496, -0.061296, -0.000100, 0.000000, 3.141593, 0.000000],accel_mss,speed_ms,0,0.000)
    |   movel(p[0.463382, -0.061277, -0.000100, 0.000000, -3.141593, 0.000000],accel_mss,speed_ms,0,0.000)
    |   movel(p[0.463281, -0.061264, -0.000100, 0.000000, -3.141593, 0.000000],accel_mss,speed_ms,0,0.000)
    |   movel(p[0.463130, -0.061217, -0.000100, 0.000000, -3.141593, 0.000000],accel_mss,speed_ms,0,0.000)
    |   movel(p[0.462961, -0.061152, -0.000100, 0.000000, 3.141593, 0.000000],accel_mss,speed_ms,0,0.000)
    |   movel(p[0.462799, -0.061074, -0.000100, 0.000000, -3.141593, 0.000000],accel_mss,speed_ms,0,0.000)
    |   movel(p[0.462544, -0.060985, -0.000100, 0.000000, -3.141593, 0.000000],accel_mss,speed_ms,0,0.000)
    |   movel(p[0.462174, -0.060934, -0.000100, 0.000000, -3.141593, 0.000000],accel_mss,speed_ms,0,0.000)
    |   movel(p[0.461680, -0.060916, -0.000100, 0.000000, -3.141593, 0.000000],accel_mss,speed_ms,0,0.000)
    |   movel(p[0.461024, -0.060931, -0.000100, 0.000000, -3.141593, 0.000000],accel_mss,speed_ms,0,blend_radius_m)
    |   movel(p[0.460407, -0.060949, -0.000100, 0.000000, -3.141593, 0.000000],accel_mss,speed_ms,0,blend_radius_m)
    |   movel(p[0.460003, -0.060937, -0.000100, 0.000000, -3.141593, 0.000000],accel_mss,speed_ms,0,0.000)
    |   movel(p[0.459761, -0.060902, -0.000100, 0.000000, -3.141593, 0.000000],accel_mss,speed_ms,0,0.000)
    |   movel(p[0.459790, -0.060774, -0.000100, 0.000000, -3.141593, 0.000000],accel_mss,speed_ms,0,0.000)
    |   movel(p[0.459883, -0.060724, -0.000100, 0.000000, 3.141593, 0.000000],accel_mss,speed_ms,0,0.000)
    |   movel(p[0.459996, -0.060690, -0.000100, 0.000000, -3.141593, 0.000000],accel_mss,speed_ms,0,0.000)
    |   movel(p[0.460111, -0.060678, -0.000100, 0.000000, -3.141593, 0.000000],accel_mss,speed_ms,0,0.000)
    |   movel(p[0.460226, -0.060667, -0.000100, 0.000000, 3.141593, 0.000000],accel_mss,speed_ms,0,0.000)
    |   movel(p[0.460339, -0.060632, -0.000100, 0.000000, -3.141593, 0.000000],accel_mss,speed_ms,0,0.000)
    |   movel(p[0.460434, -0.060580, -0.000100, 0.000000, -3.141593, 0.000000],accel_mss,speed_ms,0,0.000)
    |   movel(p[0.460551, -0.060448, -0.000100, 0.000000, -3.141593, 0.000000],accel_mss,speed_ms,0,0.000)
    |   movel(p[0.460656, -0.060363, -0.000100, 0.000000, -3.141593, 0.000000],accel_mss,speed_ms,0,0.000)
    |   movel(p[0.460782, -0.060281, -0.000100, 0.000000, -3.141593, 0.000000],accel_mss,speed_ms,0,0.000)
    |   movel(p[0.460913, -0.060213, -0.000100, 0.000000, -3.141593, 0.000000],accel_mss,speed_ms,0,0.000)
    |   movel(p[0.461405, -0.059962, -0.000100, 0.000000, -3.141593, 0.000000],accel_mss,speed_ms,0,blend_radius_m)
    |   movel(p[0.461815, -0.059696, -0.000100, 0.000000, 3.141593, 0.000000],accel_mss,speed_ms,0,0.000)
    |   movel(p[0.462241, -0.059346, -0.000100, 0.000000, -3.141593, 0.000000],accel_mss,speed_ms,0,blend_radius_m)
    |   movel(p[0.462792, -0.058822, -0.000100, 0.000000, 3.141593, 0.000000],accel_mss,speed_ms,0,blend_radius_m)
    |   movel(p[0.463472, -0.058210, -0.000100, 0.000000, -3.141593, 0.000000],accel_mss,speed_ms,0,blend_radius_m)
    |   movel(p[0.463941, -0.057973, -0.000100, 0.000000, -3.141593, 0.000000],accel_mss,speed_ms,0,blend_radius_m)
    |   movel(p[0.464300, -0.058030, -0.000100, 0.000000, -3.141593, 0.000000],accel_mss,speed_ms,0,0.000)
    |   movel(p[0.464605, -0.058353, -0.000100, 0.000000, -3.141593, 0.000000],accel_mss,speed_ms,0,0.000)
    |   movel(p[0.464881, -0.058925, -0.000100, 0.000000, -3.141593, 0.000000],accel_mss,speed_ms,0,blend_radius_m)
    |   movel(p[0.465128, -0.059615, -0.000100, 0.000000, -3.141593, 0.000000],accel_mss,speed_ms,0,blend_radius_m)
    |   movel(p[0.465307, -0.060287, -0.000100, 0.000000, -3.141593, 0.000000],accel_mss,speed_ms,0,blend_radius_m)
    |   movel(p[0.465361, -0.060784, -0.000100, 0.000000, 3.141593, 0.000000],accel_mss,speed_ms,0,0.000)
    |   movel(p[0.465379, -0.061045, -0.000100, 0.000000, -3.141593, 0.000000],accel_mss,speed_ms,0,0.000)
    |   movel(p[0.465438, -0.061214, -0.000100, 0.000000, -3.141593, 0.000000],accel_mss,speed_ms,0,0.000)
    |   movel(p[0.465553, -0.061334, -0.000100, 0.000000, -3.141593, 0.000000],accel_mss,speed_ms,0,0.000)
    |   movel(p[0.465746, -0.061432, -0.000100, 0.000000, -3.141593, 0.000000],accel_mss,speed_ms,0,0.000)
    |   movel(p[0.466123, -0.061556, -0.000100, 0.000000, -3.141593, 0.000000],accel_mss,speed_ms,0,0.000)
    |   movel(p[0.466300, -0.061537, -0.000100, 0.000000, -3.141593, 0.000000],accel_mss,speed_ms,0,0.000)
    |   movel(p[0.466410, -0.061403, -0.000100, 0.000000, 3.141593, 0.000000],accel_mss,speed_ms,0,0.000)
    |   movel(p[0.466499, -0.061036, -0.000100, 0.000000, -3.141593, 0.000000],accel_mss,speed_ms,0,0.000)
    |   movel(p[0.466514, -0.060506, -0.000100, 0.000000, -3.141593, 0.000000],accel_mss,speed_ms,0,blend_radius_m)
    |   movel(p[0.466371, -0.059685, -0.000100, 0.000000, -3.141593, 0.000000],accel_mss,speed_ms,0,blend_radius_m)
    |   movel(p[0.466160, -0.058888, -0.000100, 0.000000, 3.141593, 0.000000],accel_mss,speed_ms,0,blend_radius_m)
    |   movel(p[0.465935, -0.058472, -0.000100, 0.000000, -3.141593, 0.000000],accel_mss,speed_ms,0,0.000)
    |   movel(p[0.465675, -0.058086, -0.000100, 0.000000, -3.141593, 0.000000],accel_mss,speed_ms,0,0.000)
    |   movel(p[0.465311, -0.057373, -0.000100, 0.000000, -3.141593, 0.000000],accel_mss,speed_ms,0,blend_radius_m)
    |   movel(p[0.464973, -0.056642, -0.000100, 0.000000, -3.141593, 0.000000],accel_mss,speed_ms,0,blend_radius_m)
    |   movel(p[0.464911, -0.056349, -0.000100, 0.000000, 3.141593, 0.000000],accel_mss,speed_ms,0,0.000)
    |   movel(p[0.464921, -0.056239, -0.000100, 0.000000, -3.141593, 0.000000],accel_mss,speed_ms,0,0.000)
    |   movel(p[0.464950, -0.056123, -0.000100, 0.000000, -3.141593, 0.000000],accel_mss,speed_ms,0,0.000)
    |   movel(p[0.464993, -0.056019, -0.000100, 0.000000, -3.141593, 0.000000],accel_mss,speed_ms,0,0.000)
    |   movel(p[0.465113, -0.055845, -0.000100, 0.000000, -3.141593, 0.000000],accel_mss,speed_ms,0,0.000)
    |   movel(p[0.465238, -0.055568, -0.000100, 0.000000, -3.141593, 0.000000],accel_mss,speed_ms,0,0.000)
    |   movel(p[0.465377, -0.055232, -0.000100, 0.000000, 3.141593, 0.000000],accel_mss,speed_ms,0,0.000)
    |   movel(p[0.465516, -0.054861, -0.000100, 0.000000, -3.141593, 0.000000],accel_mss,speed_ms,0,0.000)
    |   movel(p[0.465654, -0.054495, -0.000100, 0.000000, -3.141593, 0.000000],accel_mss,speed_ms,0,0.000)
    |   movel(p[0.465790, -0.054174, -0.000100, 0.000000, -3.141593, 0.000000],accel_mss,speed_ms,0,0.000)
    |   movel(p[0.465913, -0.053913, -0.000100, 0.000000, -3.141593, 0.000000],accel_mss,speed_ms,0,0.000)
    |   movel(p[0.466037, -0.053853, -0.000100, 0.000000, -3.141593, 0.000000],accel_mss,speed_ms,0,0.000)
    |   movel(p[0.466144, -0.053981, -0.000100, 0.000000, -3.141593, 0.000000],accel_mss,speed_ms,0,0.000)
    |   movel(p[0.466265, -0.054172, -0.000100, 0.000000, -3.141593, 0.000000],accel_mss,speed_ms,0,0.000)
    |   movel(p[0.466385, -0.054412, -0.000100, 0.000000, -3.141593, 0.000000],accel_mss,speed_ms,0,0.000)
    |   movel(p[0.466566, -0.054725, -0.000100, 0.000000, -3.141593, 0.000000],accel_mss,speed_ms,0,0.000)
    |   movel(p[0.466893, -0.055158, -0.000100, 0.000000, 3.141593, 0.000000],accel_mss,speed_ms,0,blend_radius_m)
    |   movel(p[0.467291, -0.055622, -0.000100, 0.000000, -3.141593, 0.000000],accel_mss,speed_ms,0,blend_radius_m)
    |   movel(p[0.467706, -0.056051, -0.000100, 0.000000, -3.141593, 0.000000],accel_mss,speed_ms,0,blend_radius_m)
    |   movel(p[0.468694, -0.056881, -0.000100, 0.000000, -3.141593, 0.000000],accel_mss,speed_ms,0,blend_radius_m)
    |   movel(p[0.469614, -0.057384, -0.000100, 0.000000, -3.141593, 0.000000],accel_mss,speed_ms,0,blend_radius_m)
    |   movel(p[0.470598, -0.057620, -0.000100, 0.000000, -3.141593, 0.000000],accel_mss,speed_ms,0,blend_radius_m)
    |   movel(p[0.471777, -0.057634, -0.000100, 0.000000, -3.141593, 0.000000],accel_mss,speed_ms,0,blend_radius_m)
    |   movel(p[0.473069, -0.057416, -0.000100, 0.000000, -3.141593, 0.000000],accel_mss,speed_ms,0,blend_radius_m)
    |   movel(p[0.474031, -0.056974, -0.000100, 0.000000, -3.141593, 0.000000],accel_mss,speed_ms,0,blend_radius_m)
    |   movel(p[0.474645, -0.056318, -0.000100, 0.000000, -3.141593, 0.000000],accel_mss,speed_ms,0,blend_radius_m)
    |   movel(p[0.474923, -0.055471, -0.000100, 0.000000, -3.141593, 0.000000],accel_mss,speed_ms,0,blend_radius_m)
    |   movel(p[0.474946, -0.055083, -0.000100, 0.000000, -3.141593, 0.000000],accel_mss,speed_ms,0,0.000)
    |   movel(p[0.474919, -0.054836, -0.000100, 0.000000, -3.141593, 0.000000],accel_mss,speed_ms,0,0.000)
    |   movel(p[0.474836, -0.054649, -0.000100, 0.000000, -3.141593, 0.000000],accel_mss,speed_ms,0,0.000)
    |   movel(p[0.474680, -0.054470, -0.000100, 0.000000, -3.141593, 0.000000],accel_mss,speed_ms,0,0.000)
    |   movel(p[0.474476, -0.054300, -0.000100, 0.000000, -3.141593, 0.000000],accel_mss,speed_ms,0,0.000)
    |   movel(p[0.474370, -0.054271, -0.000100, 0.000000, -3.141593, 0.000000],accel_mss,speed_ms,0,0.000)
    |   movel(p[0.474268, -0.054324, -0.000100, 0.000000, -3.141593, 0.000000],accel_mss,speed_ms,0,0.000)
    |   movel(p[0.474075, -0.054545, -0.000100, 0.000000, -3.141593, 0.000000],accel_mss,speed_ms,0,0.000)
    |   movel(p[0.473962, -0.054704, -0.000100, 0.000000, -3.141593, 0.000000],accel_mss,speed_ms,0,0.000)
    |   movel(p[0.473898, -0.054846, -0.000100, 0.000000, 3.141593, 0.000000],accel_mss,speed_ms,0,0.000)
    |   movel(p[0.473884, -0.054962, -0.000100, 0.000000, 3.141593, 0.000000],accel_mss,speed_ms,0,0.000)
    |   movel(p[0.473977, -0.055623, -0.000100, 0.000000, -3.141593, 0.000000],accel_mss,speed_ms,0,blend_radius_m)
    |   movel(p[0.473290, -0.056328, -0.000100, 0.000000, -3.141593, 0.000000],accel_mss,speed_ms,0,blend_radius_m)
    |   movel(p[0.472150, -0.056906, -0.000100, 0.000000, -3.141593, 0.000000],accel_mss,speed_ms,0,blend_radius_m)
    |   movel(p[0.470974, -0.057097, -0.000100, 0.000000, 3.141593, 0.000000],accel_mss,speed_ms,0,blend_radius_m)
    |   movel(p[0.470387, -0.057058, -0.000100, 0.000000, -3.141593, 0.000000],accel_mss,speed_ms,0,blend_radius_m)
    |   movel(p[0.469879, -0.056952, -0.000100, 0.000000, -3.141593, 0.000000],accel_mss,speed_ms,0,blend_radius_m)
    |   movel(p[0.469515, -0.056804, -0.000100, 0.000000, -3.141593, 0.000000],accel_mss,speed_ms,0,0.000)
    |   movel(p[0.469411, -0.056632, -0.000100, 0.000000, -3.141593, 0.000000],accel_mss,speed_ms,0,0.000)
    |   movel(p[0.469349, -0.056523, -0.000100, 0.000000, -3.141593, 0.000000],accel_mss,speed_ms,0,0.000)
    |   movel(p[0.469199, -0.056478, -0.000100, 0.000000, -3.141593, 0.000000],accel_mss,speed_ms,0,0.000)
    |   movel(p[0.468853, -0.056330, -0.000100, 0.000000, -3.141593, 0.000000],accel_mss,speed_ms,0,0.000)
    |   movel(p[0.467795, -0.055190, -0.000100, 0.000000, -3.141593, 0.000000],accel_mss,speed_ms,0,blend_radius_m)
    |   movel(p[0.466811, -0.054046, -0.000100, 0.000000, 3.141593, 0.000000],accel_mss,speed_ms,0,blend_radius_m)
    |   movel(p[0.466321, -0.053296, -0.000100, 0.000000, -3.141593, 0.000000],accel_mss,speed_ms,0,blend_radius_m)
    |   movel(p[0.466173, -0.052959, -0.000100, 0.000000, -3.141593, 0.000000],accel_mss,speed_ms,0,0.000)
    |   movel(p[0.466058, -0.052599, -0.000100, 0.000000, -3.141593, 0.000000],accel_mss,speed_ms,0,0.000)
    |   movel(p[0.465985, -0.052243, -0.000100, 0.000000, 3.141593, 0.000000],accel_mss,speed_ms,0,0.000)
    |   movel(p[0.465961, -0.051920, -0.000100, 0.000000, -3.141593, 0.000000],accel_mss,speed_ms,0,0.000)
    |   movel(p[0.465948, -0.051608, -0.000100, 0.000000, -3.141593, 0.000000],accel_mss,speed_ms,0,0.000)
    |   movel(p[0.465908, -0.051219, -0.000100, 0.000000, 3.141593, 0.000000],accel_mss,speed_ms,0,0.000)
    |   movel(p[0.465850, -0.050819, -0.000100, 0.000000, 3.141593, 0.000000],accel_mss,speed_ms,0,0.000)
    |   movel(p[0.465781, -0.050472, -0.000100, 0.000000, -3.141593, 0.000000],accel_mss,speed_ms,0,0.000)
    |   movel(p[0.465685, -0.050012, -0.000100, 0.000000, -3.141593, 0.000000],accel_mss,speed_ms,0,0.000)
    |   movel(p[0.465675, -0.049785, -0.000100, 0.000000, -3.141593, 0.000000],accel_mss,speed_ms,0,0.000)
    |   movel(p[0.465734, -0.049633, -0.000100, 0.000000, -3.141593, 0.000000],accel_mss,speed_ms,0,0.000)
    |   movel(p[0.465878, -0.049490, -0.000100, 0.000000, 3.141593, 0.000000],accel_mss,speed_ms,0,0.000)
    |   movel(p[0.465992, -0.049418, -0.000100, 0.000000, -3.141593, 0.000000],accel_mss,speed_ms,0,0.000)
    |   movel(p[0.466107, -0.049368, -0.000100, 0.000000, -3.141593, 0.000000],accel_mss,speed_ms,0,0.000)
    |   movel(p[0.466205, -0.049344, -0.000100, 0.000000, -3.141593, 0.000000],accel_mss,speed_ms,0,0.000)
    |   movel(p[0.466337, -0.049355, -0.000100, 0.000000, -3.141593, 0.000000],accel_mss,speed_ms,0,0.000)
    |   movel(p[0.466507, -0.049227, -0.000100, 0.000000, -3.141593, 0.000000],accel_mss,speed_ms,0,0.000)
    |   movel(p[0.466710, -0.049045, -0.000100, 0.000000, -3.141593, 0.000000],accel_mss,speed_ms,0,0.000)
    |   movel(p[0.466929, -0.048816, -0.000100, 0.000000, -3.141593, 0.000000],accel_mss,speed_ms,0,0.000)
    |   movel(p[0.467341, -0.048418, -0.000100, 0.000000, 3.141593, 0.000000],accel_mss,speed_ms,0,blend_radius_m)
    |   movel(p[0.467611, -0.048348, -0.000100, 0.000000, -3.141593, 0.000000],accel_mss,speed_ms,0,0.000)
    |   movel(p[0.467849, -0.048511, -0.000100, 0.000000, -3.141593, 0.000000],accel_mss,speed_ms,0,0.000)
    |   movel(p[0.468144, -0.049050, -0.000100, 0.000000, 3.141593, 0.000000],accel_mss,speed_ms,0,blend_radius_m)
    |   movel(p[0.468269, -0.049461, -0.000100, 0.000000, -3.141593, 0.000000],accel_mss,speed_ms,0,0.000)
    |   movel(p[0.468244, -0.049843, -0.000100, 0.000000, -3.141593, 0.000000],accel_mss,speed_ms,0,0.000)
    |   movel(p[0.468058, -0.050219, -0.000100, 0.000000, -3.141593, 0.000000],accel_mss,speed_ms,0,0.000)
    |   movel(p[0.467702, -0.050617, -0.000100, 0.000000, -3.141593, 0.000000],accel_mss,speed_ms,0,blend_radius_m)
    |   movel(p[0.467451, -0.050933, -0.000100, 0.000000, -3.141593, 0.000000],accel_mss,speed_ms,0,0.000)
    |   movel(p[0.467323, -0.051294, -0.000100, 0.000000, -3.141593, 0.000000],accel_mss,speed_ms,0,0.000)
    |   movel(p[0.467354, -0.051566, -0.000100, 0.000000, -3.141593, 0.000000],accel_mss,speed_ms,0,0.000)
    |   movel(p[0.467523, -0.051678, -0.000100, 0.000000, -3.141593, 0.000000],accel_mss,speed_ms,0,0.000)
    |   movel(p[0.467639, -0.051641, -0.000100, 0.000000, -3.141593, 0.000000],accel_mss,speed_ms,0,0.000)
    |   movel(p[0.467852, -0.051475, -0.000100, 0.000000, -3.141593, 0.000000],accel_mss,speed_ms,0,0.000)
    |   movel(p[0.468096, -0.051251, -0.000100, 0.000000, -3.141593, 0.000000],accel_mss,speed_ms,0,0.000)
    |   movel(p[0.468345, -0.050986, -0.000100, 0.000000, -3.141593, 0.000000],accel_mss,speed_ms,0,0.000)
    |   movel(p[0.468754, -0.050529, -0.000100, 0.000000, -3.141593, 0.000000],accel_mss,speed_ms,0,blend_radius_m)
    |   movel(p[0.468896, -0.050427, -0.000100, 0.000000, -3.141593, 0.000000],accel_mss,speed_ms,0,0.000)
    |   movel(p[0.468998, -0.050454, -0.000100, 0.000000, -3.141593, 0.000000],accel_mss,speed_ms,0,0.000)
    |   movel(p[0.469108, -0.050648, -0.000100, 0.000000, -3.141593, 0.000000],accel_mss,speed_ms,0,0.000)
    |   movel(p[0.469178, -0.050801, -0.000100, 0.000000, -3.141593, 0.000000],accel_mss,speed_ms,0,0.000)
    |   movel(p[0.469265, -0.050968, -0.000100, 0.000000, -3.141593, 0.000000],accel_mss,speed_ms,0,0.000)
    |   movel(p[0.469354, -0.051124, -0.000100, 0.000000, -3.141593, 0.000000],accel_mss,speed_ms,0,0.000)
    |   movel(p[0.469430, -0.051239, -0.000100, 0.000000, -3.141593, 0.000000],accel_mss,speed_ms,0,0.000)
    |   movel(p[0.469498, -0.051385, -0.000100, 0.000000, -3.141593, 0.000000],accel_mss,speed_ms,0,0.000)
    |   movel(p[0.469507, -0.051549, -0.000100, 0.000000, -3.141593, 0.000000],accel_mss,speed_ms,0,0.000)
    |   movel(p[0.469456, -0.051761, -0.000100, 0.000000, -3.141593, 0.000000],accel_mss,speed_ms,0,0.000)
    |   movel(p[0.469331, -0.052064, -0.000100, 0.000000, -3.141593, 0.000000],accel_mss,speed_ms,0,0.000)
    |   movel(p[0.469212, -0.052308, -0.000100, 0.000000, -3.141593, 0.000000],accel_mss,speed_ms,0,0.000)
    |   movel(p[0.469078, -0.052554, -0.000100, 0.000000, 3.141593, 0.000000],accel_mss,speed_ms,0,0.000)
    |   movel(p[0.468948, -0.052768, -0.000100, 0.000000, 3.141593, 0.000000],accel_mss,speed_ms,0,0.000)
    |   movel(p[0.468849, -0.052903, -0.000100, 0.000000, -3.141593, 0.000000],accel_mss,speed_ms,0,0.000)
    |   movel(p[0.468771, -0.053025, -0.000100, 0.000000, -3.141593, 0.000000],accel_mss,speed_ms,0,0.000)
    |   movel(p[0.468714, -0.053183, -0.000100, 0.000000, -3.141593, 0.000000],accel_mss,speed_ms,0,0.000)
    |   movel(p[0.468683, -0.053351, -0.000100, 0.000000, -3.141593, 0.000000],accel_mss,speed_ms,0,0.000)
    |   movel(p[0.468687, -0.053503, -0.000100, 0.000000, -3.141593, 0.000000],accel_mss,speed_ms,0,0.000)
    |   movel(p[0.468732, -0.053680, -0.000100, 0.000000, -3.141593, 0.000000],accel_mss,speed_ms,0,0.000)
    |   movel(p[0.468812, -0.053779, -0.000100, 0.000000, -3.141593, 0.000000],accel_mss,speed_ms,0,0.000)
    |   movel(p[0.468944, -0.053823, -0.000100, 0.000000, -3.141593, 0.000000],accel_mss,speed_ms,0,0.000)
    |   movel(p[0.469170, -0.053822, -0.000100, 0.000000, 3.141593, 0.000000],accel_mss,speed_ms,0,0.000)
    |   movel(p[0.469361, -0.053787, -0.000100, 0.000000, -3.141593, 0.000000],accel_mss,speed_ms,0,0.000)
    |   movel(p[0.469578, -0.053704, -0.000100, 0.000000, 3.141593, 0.000000],accel_mss,speed_ms,0,0.000)
    |   movel(p[0.469787, -0.053591, -0.000100, 0.000000, -3.141593, 0.000000],accel_mss,speed_ms,0,0.000)
    |   movel(p[0.469953, -0.053463, -0.000100, 0.000000, -3.141593, 0.000000],accel_mss,speed_ms,0,0.000)
    |   movel(p[0.470147, -0.053296, -0.000100, 0.000000, -3.141593, 0.000000],accel_mss,speed_ms,0,0.000)
    |   movel(p[0.470279, -0.053233, -0.000100, 0.000000, -3.141593, 0.000000],accel_mss,speed_ms,0,0.000)
    |   movel(p[0.470397, -0.053243, -0.000100, 0.000000, 3.141593, 0.000000],accel_mss,speed_ms,0,0.000)
    |   movel(p[0.470532, -0.053325, -0.000100, 0.000000, -3.141593, 0.000000],accel_mss,speed_ms,0,0.000)
    |   movel(p[0.470619, -0.053411, -0.000100, 0.000000, -3.141593, 0.000000],accel_mss,speed_ms,0,0.000)
    |   movel(p[0.470694, -0.053512, -0.000100, 0.000000, -3.141593, 0.000000],accel_mss,speed_ms,0,0.000)
    |   movel(p[0.470745, -0.053613, -0.000100, 0.000000, -3.141593, 0.000000],accel_mss,speed_ms,0,0.000)
    |   movel(p[0.470974, -0.054122, -0.000100, 0.000000, -3.141593, 0.000000],accel_mss,speed_ms,0,blend_radius_m)
    |   movel(p[0.471724, -0.054581, -0.000100, 0.000000, -3.141593, 0.000000],accel_mss,speed_ms,0,blend_radius_m)
    |   movel(p[0.472622, -0.054920, -0.000100, 0.000000, -3.141593, 0.000000],accel_mss,speed_ms,0,blend_radius_m)
    |   movel(p[0.473386, -0.054984, -0.000100, 0.000000, -3.141593, 0.000000],accel_mss,speed_ms,0,blend_radius_m)
    |   movel(p[0.473518, -0.054959, -0.000100, 0.000000, -3.141593, 0.000000],accel_mss,speed_ms,0,0.000)
    |   movel(p[0.473463, -0.054861, -0.000100, 0.000000, -3.141593, 0.000000],accel_mss,speed_ms,0,0.000)
    |   movel(p[0.473217, -0.054748, -0.000100, 0.000000, -3.141593, 0.000000],accel_mss,speed_ms,0,0.000)
    |   movel(p[0.473004, -0.054637, -0.000100, 0.000000, -3.141593, 0.000000],accel_mss,speed_ms,0,0.000)
    |   movel(p[0.472749, -0.054466, -0.000100, 0.000000, 3.141593, 0.000000],accel_mss,speed_ms,0,0.000)
    |   movel(p[0.472495, -0.054270, -0.000100, 0.000000, -3.141593, 0.000000],accel_mss,speed_ms,0,0.000)
    |   movel(p[0.472283, -0.054077, -0.000100, 0.000000, 3.141593, 0.000000],accel_mss,speed_ms,0,0.000)
    |   movel(p[0.471978, -0.053735, -0.000100, 0.000000, -3.141593, 0.000000],accel_mss,speed_ms,0,0.000)
    |   movel(p[0.471747, -0.053392, -0.000100, 0.000000, -3.141593, 0.000000],accel_mss,speed_ms,0,0.000)
    |   movel(p[0.471496, -0.052895, -0.000100, 0.000000, -3.141593, 0.000000],accel_mss,speed_ms,0,blend_radius_m)
    |   movel(p[0.471058, -0.051903, -0.000100, 0.000000, -3.141593, 0.000000],accel_mss,speed_ms,0,blend_radius_m)
    |   movel(p[0.470604, -0.050882, -0.000100, 0.000000, -3.141593, 0.000000],accel_mss,speed_ms,0,blend_radius_m)
    |   movel(p[0.470223, -0.050082, -0.000100, 0.000000, -3.141593, 0.000000],accel_mss,speed_ms,0,blend_radius_m)
    |   movel(p[0.469901, -0.049469, -0.000100, 0.000000, -3.141593, 0.000000],accel_mss,speed_ms,0,blend_radius_m)
    |   movel(p[0.469638, -0.049053, -0.000100, 0.000000, -3.141593, 0.000000],accel_mss,speed_ms,0,0.000)
    |   movel(p[0.469506, -0.048865, -0.000100, 0.000000, -3.141593, 0.000000],accel_mss,speed_ms,0,0.000)
    |   movel(p[0.469379, -0.048669, -0.000100, 0.000000, -3.141593, 0.000000],accel_mss,speed_ms,0,0.000)
    |   movel(p[0.469271, -0.048494, -0.000100, 0.000000, -3.141593, 0.000000],accel_mss,speed_ms,0,0.000)
    |   movel(p[0.469211, -0.048378, -0.000100, 0.000000, -3.141593, 0.000000],accel_mss,speed_ms,0,0.000)
    |   movel(p[0.469152, -0.048262, -0.000100, 0.000000, -3.141593, 0.000000],accel_mss,speed_ms,0,0.000)
    |   movel(p[0.469051, -0.048087, -0.000100, 0.000000, -3.141593, 0.000000],accel_mss,speed_ms,0,0.000)
    |   movel(p[0.468932, -0.047892, -0.000100, 0.000000, 3.141593, 0.000000],accel_mss,speed_ms,0,0.000)
    |   movel(p[0.468812, -0.047703, -0.000100, 0.000000, -3.141593, 0.000000],accel_mss,speed_ms,0,0.000)
    |   movel(p[0.468688, -0.047509, -0.000100, 0.000000, -3.141593, 0.000000],accel_mss,speed_ms,0,0.000)
    |   movel(p[0.468563, -0.047297, -0.000100, 0.000000, 3.141593, 0.000000],accel_mss,speed_ms,0,0.000)
    |   movel(p[0.468453, -0.047099, -0.000100, 0.000000, -3.141593, 0.000000],accel_mss,speed_ms,0,0.000)
    |   movel(p[0.468380, -0.046953, -0.000100, 0.000000, 3.141593, 0.000000],accel_mss,speed_ms,0,0.000)
    |   movel(p[0.468224, -0.046698, -0.000100, 0.000000, -3.141593, 0.000000],accel_mss,speed_ms,0,0.000)
    |   movel(p[0.467988, -0.046454, -0.000100, 0.000000, -3.141593, 0.000000],accel_mss,speed_ms,0,0.000)
    |   movel(p[0.467659, -0.046206, -0.000100, 0.000000, -3.141593, 0.000000],accel_mss,speed_ms,0,0.000)
    |   movel(p[0.467213, -0.045939, -0.000100, 0.000000, -3.141593, 0.000000],accel_mss,speed_ms,0,blend_radius_m)
    |   movel(p[0.466657, -0.045750, -0.000100, 0.000000, -3.141593, 0.000000],accel_mss,speed_ms,0,blend_radius_m)
    |   movel(p[0.465857, -0.045683, -0.000100, 0.000000, -3.141593, 0.000000],accel_mss,speed_ms,0,blend_radius_m)
    |   movel(p[0.464953, -0.045734, -0.000100, 0.000000, -3.141593, 0.000000],accel_mss,speed_ms,0,blend_radius_m)
    |   movel(p[0.464062, -0.045903, -0.000100, 0.000000, -3.141593, 0.000000],accel_mss,speed_ms,0,blend_radius_m)
    |   movel(p[0.463226, -0.046106, -0.000100, 0.000000, -3.141593, 0.000000],accel_mss,speed_ms,0,blend_radius_m)
    |   movel(p[0.462980, -0.046070, -0.000100, 0.000000, -3.141593, 0.000000],accel_mss,speed_ms,0,0.000)
    |   movel(p[0.462864, -0.045882, -0.000100, 0.000000, 3.141593, 0.000000],accel_mss,speed_ms,0,0.000)
    |   movel(p[0.462854, -0.045223, -0.000100, 0.000000, -3.141593, 0.000000],accel_mss,speed_ms,0,blend_radius_m)
    |   movel(p[0.462863, -0.044770, -0.000100, 0.000000, 3.141593, 0.000000],accel_mss,speed_ms,0,0.000)
    |   movel(p[0.462871, -0.044317, -0.000100, 0.000000, -3.141593, 0.000000],accel_mss,speed_ms,0,0.000)
    |   movel(p[0.462440, -0.043888, -0.000100, 0.000000, 3.141593, 0.000000],accel_mss,speed_ms,0,blend_radius_m)
    |   movel(p[0.462008, -0.043460, -0.000100, 0.000000, -3.141593, 0.000000],accel_mss,speed_ms,0,blend_radius_m)
    |   movel(p[0.461477, -0.042943, -0.000100, 0.000000, -3.141593, 0.000000],accel_mss,speed_ms,0,blend_radius_m)
    |   movel(p[0.461246, -0.042775, -0.000100, 0.000000, -3.141593, 0.000000],accel_mss,speed_ms,0,0.000)
    |   movel(p[0.461090, -0.042764, -0.000100, 0.000000, -3.141593, 0.000000],accel_mss,speed_ms,0,0.000)
    |   movel(p[0.460943, -0.042875, -0.000100, 0.000000, -3.141593, 0.000000],accel_mss,speed_ms,0,0.000)
    |   movel(p[0.460861, -0.043041, -0.000100, 0.000000, -3.141593, 0.000000],accel_mss,speed_ms,0,0.000)
    |   movel(p[0.460796, -0.043332, -0.000100, 0.000000, -3.141593, 0.000000],accel_mss,speed_ms,0,0.000)
    |   movel(p[0.460751, -0.043687, -0.000100, 0.000000, -3.141593, 0.000000],accel_mss,speed_ms,0,0.000)
    |   movel(p[0.460735, -0.044075, -0.000100, 0.000000, -3.141593, 0.000000],accel_mss,speed_ms,0,0.000)
    |   movel(p[0.460732, -0.044446, -0.000100, 0.000000, -3.141593, 0.000000],accel_mss,speed_ms,0,0.000)
    |   movel(p[0.460728, -0.044792, -0.000100, 0.000000, -3.141593, 0.000000],accel_mss,speed_ms,0,0.000)
    |   movel(p[0.460724, -0.045083, -0.000100, 0.000000, -3.141593, 0.000000],accel_mss,speed_ms,0,0.000)
    |   movel(p[0.460720, -0.045212, -0.000100, 0.000000, -3.141593, 0.000000],accel_mss,speed_ms,0,0.000)
    |   movel(p[0.460666, -0.045308, -0.000100, 0.000000, -3.141593, 0.000000],accel_mss,speed_ms,0,0.000)
    |   movel(p[0.460529, -0.045360, -0.000100, 0.000000, 3.141593, 0.000000],accel_mss,speed_ms,0,0.000)
    |   movel(p[0.460275, -0.045372, -0.000100, 0.000000, -3.141593, 0.000000],accel_mss,speed_ms,0,0.000)
    |   speed_ms    = 0.050
    |   movel(p[0.460275, -0.045372, 0.003000, 0.000000, -3.141593, 0.000000],accel_mss,speed_ms,0,blend_radius_m)
    |   speed_ms    = 1.000
    |   movel(p[0.460275, -0.045372, 0.015000, 0.000000, -3.141593, 0.000000],accel_mss,speed_ms,0,blend_radius_m)
    |   movel(p[0.386812, -0.046962, 0.015000, 0.000000, 3.141593, 0.000000],accel_mss,speed_ms,0,blend_radius_m)
    |   movel(p[0.386812, -0.046962, 0.003000, 0.000000, 3.141593, 0.000000],accel_mss,speed_ms,0,blend_radius_m)
    |   speed_ms    = 0.050
    |   movel(p[0.386812, -0.046962, -0.000100, 0.000000, 3.141593, 0.000000],accel_mss,speed_ms,0,blend_radius_m)
    |   speed_ms    = 0.083
    |   movel(p[0.386795, -0.048666, -0.000100, 0.000000, -3.141593, 0.000000],accel_mss,speed_ms,0,blend_radius_m)
    |   movel(p[0.386646, -0.050103, -0.000100, 0.000000, -3.141593, 0.000000],accel_mss,speed_ms,0,blend_radius_m)
    |   movel(p[0.386574, -0.050560, -0.000100, 0.000000, -3.141593, 0.000000],accel_mss,speed_ms,0,0.000)
    |   movel(p[0.386497, -0.051065, -0.000100, 0.000000, -3.141593, 0.000000],accel_mss,speed_ms,0,blend_radius_m)
